LIN {X 0,Y 424.552,Z 355.445,A -85,B 0,C 180,E1 -10322.013,E2 -10322.013} C_VEL
LIN {X 0,Y 427.893,Z 370.379,A -85,B 0,C 180,E1 -10322.491,E2 -10322.491} C_VEL
LIN {X 0,Y 426.261,Z 483.338,A -85,B 0,C 180,E1 -10324.453,E2 -10324.453} C_VEL
LIN {X 0,Y 425.683,Z 497.997,A -85,B 0,C 180,E1 -10324.903,E2 -10324.903} C_VEL
LIN {X 0,Y 424.866,Z 511.461,A -85,B 0,C 180,E1 -10325.503,E2 -10325.503} C_VEL
LIN {X 0,Y 424.074,Z 524.723,A -85,B 0,C 180,E1 -10326.304,E2 -10326.304} C_VEL
LIN {X 0,Y 423.002,Z 537.419,A -85,B 0,C 180,E1 -10327.276,E2 -10327.276} C_VEL
LIN {X 0,Y 421.99,Z 548.966,A -85,B 0,C 180,E1 -10328.378,E2 -10328.378} C_VEL
LIN {X 0,Y 420.973,Z 560.52,A -85,B 0,C 180,E1 -10329.732,E2 -10329.732} C_VEL
LIN {X 0,Y 419.941,Z 570.774,A -85,B 0,C 180,E1 -10331.206,E2 -10331.206} C_VEL
LIN {X 0,Y 419.14,Z 579.23,A -85,B 0,C 180,E1 -10332.682,E2 -10332.682} C_VEL
LIN {X 0,Y 418.394,Z 587.297,A -85,B 0,C 180,E1 -10334.409,E2 -10334.409} C_VEL
LIN {X 0,Y 418.003,Z 591.69,A -85,B 0,C 180,E1 -10335.539,E2 -10335.539} C_VEL
LIN {X 0,Y 417.168,Z 594.262,A -85,B 0,C 180,E1 -10336.26,E2 -10336.26} C_VEL
LIN {X 0,Y 414.047,Z 598.094,A -85,B 0,C 180,E1 -10337.445,E2 -10337.445} C_VEL
LIN {X 0,Y 411.436,Z 600.721,A -85,B 0,C 180,E1 -10338.424,E2 -10338.424} C_VEL
LIN {X 0,Y 410.257,Z 602.444,A -85,B 0,C 180,E1 -10339.2,E2 -10339.2} C_VEL
LIN {X 0,Y 410.128,Z 602.917,A -85,B 0,C 180,E1 -10339.467,E2 -10339.467} C_VEL
LIN {X 0,Y 409.996,Z 605.551,A -85,B 0,C 180,E1 -10341.125,E2 -10341.125} C_VEL
LIN {X 0,Y 409.948,Z 607.379,A -85,B 0,C 180,E1 -10343.108,E2 -10343.108} C_VEL
LIN {X 0,Y 409.945,Z 607.876,A -85,B 0,C 180,E1 -10345.083,E2 -10345.083} C_VEL
LIN {X 0,Y 409.955,Z 607.058,A -85,B 0,C 180,E1 -10347.052,E2 -10347.052} C_VEL
LIN {X 0,Y 410.017,Z 606.153,A -85,B 0,C 180,E1 -10348.035,E2 -10348.035} C_VEL
LIN {X 0,Y 409.997,Z 603.337,A -85,B 0,C 180,E1 -10350,E2 -10350} C_VEL
LIN {X 0,Y 410.238,Z 600.322,A -85,B 0,C 180,E1 -10351.472,E2 -10351.472} C_VEL
LIN {X 0,Y 410.609,Z 594.902,A -85,B 0,C 180,E1 -10353.434,E2 -10353.434} C_VEL
LIN {X 0,Y 411.027,Z 589.771,A -85,B 0,C 180,E1 -10354.904,E2 -10354.904} C_VEL
LIN {X 0,Y 411.731,Z 582.375,A -85,B 0,C 180,E1 -10356.616,E2 -10356.616} C_VEL
LIN {X 0,Y 412.149,Z 576.039,A -85,B 0,C 180,E1 -10357.841,E2 -10357.841} C_VEL
LIN {X 0,Y 412.694,Z 568.684,A -85,B 0,C 180,E1 -10359.063,E2 -10359.063} C_VEL
LIN {X 0,Y 413.77,Z 558.137,A -85,B 0,C 180,E1 -10360.521,E2 -10360.521} C_VEL
LIN {X 0,Y 414.662,Z 547.501,A -85,B 0,C 180,E1 -10361.735,E2 -10361.735} C_VEL
LIN {X 0,Y 415.578,Z 535.885,A -85,B 0,C 180,E1 -10362.824,E2 -10362.824} C_VEL
LIN {X 0,Y 416.477,Z 523.1,A -85,B 0,C 180,E1 -10363.79,E2 -10363.79} C_VEL
LIN {X 0,Y 417.318,Z 509.784,A -85,B 0,C 180,E1 -10364.57,E2 -10364.57} C_VEL
LIN {X 0,Y 417.971,Z 495.947,A -85,B 0,C 180,E1 -10365.17,E2 -10365.17} C_VEL
LIN {X 0,Y 418.364,Z 482.792,A -85,B 0,C 180,E1 -10365.561,E2 -10365.561} C_VEL
LIN {X 0,Y 419.945,Z 370.675,A -85,B 0,C 180,E1 -10367.508,E2 -10367.508} C_VEL
LIN {X 0,Y 415.529,Z 350.853,A -85,B 0,C 180,E1 -10368.102,E2 -10368.102} C_VEL
LIN {X 0,Y 414.038,Z 346.546,A -85,B 0,C 180,E1 -10368.292,E2 -10368.292} C_VEL
LIN {X 0,Y 411.331,Z 333.524,A -85,B 0,C 180,E1 -10371.289,E2 -10371.289} C_VEL
LIN {X 0,Y 411.216,Z 332.89,A -85,B 0,C 180,E1 -10371.493,E2 -10371.493} C_VEL
LIN {X 0,Y 411.19,Z 332.895,A -85,B 0,C 180,E1 -10375.058,E2 -10375.058} C_VEL
LIN {X 0,Y 411.171,Z 332.896,A -85,B 0,C 180,E1 -10378.594,E2 -10378.594} C_VEL
LIN {X 0,Y 411.156,Z 332.893,A -85,B 0,C 180,E1 -10381.998,E2 -10381.998} C_VEL
LIN {X 0,Y 411.202,Z 332.89,A -85,B 0,C 180,E1 -10384.876,E2 -10384.876} C_VEL
LIN {X 0,Y 411.188,Z 332.889,A -85,B 0,C 180,E1 -10388.165,E2 -10388.165} C_VEL
LIN {X 0,Y 411.161,Z 332.889,A -85,B 0,C 180,E1 -10391.808,E2 -10391.808} C_VEL
LIN {X 0,Y 411.176,Z 332.887,A -85,B 0,C 180,E1 -10395.509,E2 -10395.509} C_VEL
LIN {X 0,Y 411.148,Z 332.894,A -85,B 0,C 180,E1 -10398.775,E2 -10398.775} C_VEL
LIN {X 0,Y 411.18,Z 332.889,A -85,B 0,C 180,E1 -10402.024,E2 -10402.024} C_VEL
LIN {X 0,Y 411.204,Z 332.887,A -85,B 0,C 180,E1 -10405.123,E2 -10405.123} C_VEL
LIN {X 0,Y 411.162,Z 332.886,A -85,B 0,C 180,E1 -10408.002,E2 -10408.002} C_VEL
LIN {X 0,Y 411.172,Z 332.887,A -85,B 0,C 180,E1 -10411.406,E2 -10411.406} C_VEL
LIN {X 0,Y 411.191,Z 332.889,A -85,B 0,C 180,E1 -10414.941,E2 -10414.941} C_VEL
LIN {X 0,Y 411.205,Z 332.883,A -85,B 0,C 180,E1 -10417.913,E2 -10417.913} C_VEL
LIN {X 0,Y 411.216,Z 332.876,A -85,B 0,C 180,E1 -10421.051,E2 -10421.051} C_VEL
LIN {X 0,Y 411.213,Z 332.889,A -85,B 0,C 180,E1 -10424.13,E2 -10424.13} C_VEL
LIN {X 0,Y 411.307,Z 332.864,A -85,B 0,C 180,E1 -10427.165,E2 -10427.165} C_VEL
LIN {X 0,Y 411.293,Z 332.86,A -85,B 0,C 180,E1 -10430.161,E2 -10430.161} C_VEL
LIN {X 0,Y 411.395,Z 332.861,A -85,B 0,C 180,E1 -10433.132,E2 -10433.132} C_VEL
LIN {X 0,Y 411.299,Z 332.872,A -85,B 0,C 180,E1 -10435.099,E2 -10435.099} C_VEL
LIN {X 0,Y 411.512,Z 332.851,A -85,B 0,C 180,E1 -10438.042,E2 -10438.042} C_VEL
LIN {X 0,Y 411.44,Z 332.851,A -85,B 0,C 180,E1 -10440.978,E2 -10440.978} C_VEL
LIN {X 0,Y 411.434,Z 332.857,A -85,B 0,C 180,E1 -10442.937,E2 -10442.937} C_VEL
LIN {X 0,Y 411.436,Z 332.857,A -85,B 0,C 180,E1 -10445.882,E2 -10445.882} C_VEL
LIN {X 0,Y 411.321,Z 332.87,A -85,B 0,C 180,E1 -10448.846,E2 -10448.846} C_VEL
LIN {X 0,Y 411.286,Z 332.879,A -85,B 0,C 180,E1 -10451.832,E2 -10451.832} C_VEL
LIN {X 0,Y 411.262,Z 332.876,A -85,B 0,C 180,E1 -10454.852,E2 -10454.852} C_VEL
LIN {X 0,Y 411.253,Z 332.882,A -85,B 0,C 180,E1 -10457.915,E2 -10457.915} C_VEL
LIN {X 0,Y 411.199,Z 332.886,A -85,B 0,C 180,E1 -10461.034,E2 -10461.034} C_VEL
LIN {X 0,Y 411.22,Z 332.886,A -85,B 0,C 180,E1 -10464.216,E2 -10464.216} C_VEL
LIN {X 0,Y 411.243,Z 332.885,A -85,B 0,C 180,E1 -10467.479,E2 -10467.479} C_VEL
LIN {X 0,Y 411.191,Z 332.889,A -85,B 0,C 180,E1 -10470.847,E2 -10470.847} C_VEL
LIN {X 0,Y 411.208,Z 332.888,A -85,B 0,C 180,E1 -10474.333,E2 -10474.333} C_VEL
LIN {X 0,Y 411.202,Z 332.889,A -85,B 0,C 180,E1 -10477.973,E2 -10477.973} C_VEL
LIN {X 0,Y 411.185,Z 332.89,A -85,B 0,C 180,E1 -10480.504,E2 -10480.504} C_VEL
LIN {X 0,Y 411.175,Z 332.894,A -85,B 0,C 180,E1 -10483.133,E2 -10483.133} C_VEL
LIN {X 0,Y 411.169,Z 332.894,A -85,B 0,C 180,E1 -10485.881,E2 -10485.881} C_VEL
LIN {X 0,Y 411.164,Z 332.892,A -85,B 0,C 180,E1 -10488.771,E2 -10488.771} C_VEL
LIN {X 0,Y 411.2,Z 332.893,A -85,B 0,C 180,E1 -10492.027,E2 -10492.027} C_VEL
LIN {X 0,Y 411.207,Z 332.893,A -85,B 0,C 180,E1 -10495.666,E2 -10495.666} C_VEL
LIN {X 0,Y 411.192,Z 332.892,A -85,B 0,C 180,E1 -10499.152,E2 -10499.152} C_VEL
LIN {X 0,Y 411.25,Z 333.05,A -85,B 0,C 180,E1 -10500.009,E2 -10500.009} C_VEL
LIN {X 0,Y 414.199,Z 346.153,A -85,B 0,C 180,E1 -10502.734,E2 -10502.734} C_VEL
LIN {X 0,Y 415.494,Z 353.398,A -85,B 0,C 180,E1 -10504.179,E2 -10504.179} C_VEL
LIN {X 0,Y 414.54,Z 367.529,A -85,B 0,C 180,E1 -10506.768,E2 -10506.768} C_VEL
LIN {X 0,Y 419.74,Z 398.333,A -85,B 0,C 180,E1 -10507.617,E2 -10507.617} C_VEL
LIN {X 0,Y 418.158,Z 504.873,A -85,B 0,C 180,E1 -10509.461,E2 -10509.461} C_VEL
LIN {X 0,Y 417.629,Z 519.149,A -85,B 0,C 180,E1 -10509.883,E2 -10509.883} C_VEL
LIN {X 0,Y 416.866,Z 532.72,A -85,B 0,C 180,E1 -10510.475,E2 -10510.475} C_VEL
LIN {X 0,Y 415.995,Z 546.287,A -85,B 0,C 180,E1 -10511.277,E2 -10511.277} C_VEL
LIN {X 0,Y 415.02,Z 559.153,A -85,B 0,C 180,E1 -10512.253,E2 -10512.253} C_VEL
LIN {X 0,Y 413.988,Z 570.843,A -85,B 0,C 180,E1 -10513.353,E2 -10513.353} C_VEL
LIN {X 0,Y 412.966,Z 582.538,A -85,B 0,C 180,E1 -10514.705,E2 -10514.705} C_VEL
LIN {X 0,Y 412.077,Z 592.992,A -85,B 0,C 180,E1 -10516.186,E2 -10516.186} C_VEL
LIN {X 0,Y 411.388,Z 601.614,A -85,B 0,C 180,E1 -10517.67,E2 -10517.67} C_VEL
LIN {X 0,Y 410.758,Z 609.847,A -85,B 0,C 180,E1 -10519.401,E2 -10519.401} C_VEL
LIN {X 0,Y 410.344,Z 616.475,A -85,B 0,C 180,E1 -10521.133,E2 -10521.133} C_VEL
LIN {X 0,Y 410.158,Z 622.354,A -85,B 0,C 180,E1 -10523.111,E2 -10523.111} C_VEL
LIN {X 0,Y 409.988,Z 626.639,A -85,B 0,C 180,E1 -10525.083,E2 -10525.083} C_VEL
LIN {X 0,Y 409.923,Z 629.47,A -85,B 0,C 180,E1 -10527.052,E2 -10527.052} C_VEL
LIN {X 0,Y 409.933,Z 630.928,A -85,B 0,C 180,E1 -10529.018,E2 -10529.018} C_VEL
LIN {X 0,Y 409.933,Z 631.045,A -85,B 0,C 180,E1 -10530.982,E2 -10530.982} C_VEL
LIN {X 0,Y 409.92,Z 629.831,A -85,B 0,C 180,E1 -10532.948,E2 -10532.948} C_VEL
LIN {X 0,Y 409.988,Z 627.259,A -85,B 0,C 180,E1 -10534.917,E2 -10534.917} C_VEL
LIN {X 0,Y 410.156,Z 623.241,A -85,B 0,C 180,E1 -10536.889,E2 -10536.889} C_VEL
LIN {X 0,Y 410.4,Z 617.672,A -85,B 0,C 180,E1 -10538.866,E2 -10538.866} C_VEL
LIN {X 0,Y 410.797,Z 611.402,A -85,B 0,C 180,E1 -10540.598,E2 -10540.598} C_VEL
LIN {X 0,Y 411.586,Z 603.609,A -85,B 0,C 180,E1 -10542.324,E2 -10542.324} C_VEL
LIN {X 0,Y 412.228,Z 595.485,A -85,B 0,C 180,E1 -10543.809,E2 -10543.809} C_VEL
LIN {X 0,Y 413.194,Z 585.715,A -85,B 0,C 180,E1 -10545.286,E2 -10545.286} C_VEL
LIN {X 0,Y 414.288,Z 574.884,A -85,B 0,C 180,E1 -10546.635,E2 -10546.635} C_VEL
LIN {X 0,Y 415.564,Z 562.897,A -85,B 0,C 180,E1 -10547.85,E2 -10547.85} C_VEL
LIN {X 0,Y 416.547,Z 551.215,A -85,B 0,C 180,E1 -10548.816,E2 -10548.816} C_VEL
LIN {X 0,Y 417.55,Z 538.211,A -85,B 0,C 180,E1 -10549.672,E2 -10549.672} C_VEL
LIN {X 0,Y 418.434,Z 524.264,A -85,B 0,C 180,E1 -10550.365,E2 -10550.365} C_VEL
LIN {X 0,Y 419.169,Z 510.595,A -85,B 0,C 180,E1 -10550.84,E2 -10550.84} C_VEL
LIN {X 0,Y 419.577,Z 495.358,A -85,B 0,C 180,E1 -10551.173,E2 -10551.173} C_VEL
LIN {X 0,Y 421.022,Z 397.613,A -85,B 0,C 180,E1 -10552.873,E2 -10552.873} C_VEL
LIN {X 0,Y 417.283,Z 377.293,A -85,B 0,C 180,E1 -10553.484,E2 -10553.484} C_VEL
LIN {X 0,Y 415.256,Z 367.358,A -85,B 0,C 180,E1 -10553.827,E2 -10553.827} C_VEL
LIN {X 0,Y 416.244,Z 355.506,A -85,B 0,C 180,E1 -10556.04,E2 -10556.04} C_VEL
LIN {X 0,Y 414.321,Z 345.621,A -85,B 0,C 180,E1 -10558.108,E2 -10558.108} C_VEL
LIN {X 0,Y 411.205,Z 332.882,A -85,B 0,C 180,E1 -10560.955,E2 -10560.955} C_VEL
LIN {X 0,Y 411.207,Z 332.89,A -85,B 0,C 180,E1 -10564.334,E2 -10564.334} C_VEL
LIN {X 0,Y 411.195,Z 332.887,A -85,B 0,C 180,E1 -10567.974,E2 -10567.974} C_VEL
LIN {X 0,Y 411.165,Z 332.891,A -85,B 0,C 180,E1 -10571.229,E2 -10571.229} C_VEL
LIN {X 0,Y 411.177,Z 332.895,A -85,B 0,C 180,E1 -10574.491,E2 -10574.491} C_VEL
LIN {X 0,Y 411.179,Z 332.89,A -85,B 0,C 180,E1 -10578.195,E2 -10578.195} C_VEL
LIN {X 0,Y 411.224,Z 332.883,A -85,B 0,C 180,E1 -10580.777,E2 -10580.777} C_VEL
LIN {X 0,Y 411.199,Z 332.89,A -85,B 0,C 180,E1 -10584.472,E2 -10584.472} C_VEL
LIN {X 0,Y 411.209,Z 332.885,A -85,B 0,C 180,E1 -10586.874,E2 -10586.874} C_VEL
LIN {X 0,Y 411.215,Z 332.887,A -85,B 0,C 180,E1 -10590.65,E2 -10590.65} C_VEL
LIN {X 0,Y 411.198,Z 332.885,A -85,B 0,C 180,E1 -10593.617,E2 -10593.617} C_VEL
LIN {X 0,Y 411.199,Z 332.884,A -85,B 0,C 180,E1 -10596.852,E2 -10596.852} C_VEL
LIN {X 0,Y 411.218,Z 332.889,A -85,B 0,C 180,E1 -10600.051,E2 -10600.051} C_VEL
LIN {X 0,Y 411.266,Z 332.875,A -85,B 0,C 180,E1 -10603.132,E2 -10603.132} C_VEL
LIN {X 0,Y 411.309,Z 332.866,A -85,B 0,C 180,E1 -10606.896,E2 -10606.896} C_VEL
LIN {X 0,Y 411.294,Z 332.876,A -85,B 0,C 180,E1 -10610.162,E2 -10610.162} C_VEL
LIN {X 0,Y 411.396,Z 332.86,A -85,B 0,C 180,E1 -10613.132,E2 -10613.132} C_VEL
LIN {X 0,Y 411.298,Z 332.874,A -85,B 0,C 180,E1 -10615.099,E2 -10615.099} C_VEL
LIN {X 0,Y 411.506,Z 332.85,A -85,B 0,C 180,E1 -10618.043,E2 -10618.043} C_VEL
LIN {X 0,Y 411.381,Z 332.86,A -85,B 0,C 180,E1 -10620.979,E2 -10620.979} C_VEL
LIN {X 0,Y 411.45,Z 332.852,A -85,B 0,C 180,E1 -10622.938,E2 -10622.938} C_VEL
LIN {X 0,Y 411.394,Z 332.854,A -85,B 0,C 180,E1 -10626.478,E2 -10626.478} C_VEL
LIN {X 0,Y 411.321,Z 332.871,A -85,B 0,C 180,E1 -10628.846,E2 -10628.846} C_VEL
LIN {X 0,Y 411.287,Z 332.873,A -85,B 0,C 180,E1 -10631.833,E2 -10631.833} C_VEL
LIN {X 0,Y 411.234,Z 332.882,A -85,B 0,C 180,E1 -10634.854,E2 -10634.854} C_VEL
LIN {X 0,Y 411.198,Z 332.891,A -85,B 0,C 180,E1 -10637.918,E2 -10637.918} C_VEL
LIN {X 0,Y 411.19,Z 332.883,A -85,B 0,C 180,E1 -10641.035,E2 -10641.035} C_VEL
LIN {X 0,Y 411.194,Z 332.884,A -85,B 0,C 180,E1 -10644.218,E2 -10644.218} C_VEL
LIN {X 0,Y 411.148,Z 332.896,A -85,B 0,C 180,E1 -10647.486,E2 -10647.486} C_VEL
LIN {X 0,Y 411.195,Z 332.87,A -85,B 0,C 180,E1 -10649.714,E2 -10649.714} C_VEL
LIN {X 0,Y 411.207,Z 332.887,A -85,B 0,C 180,E1 -10653.156,E2 -10653.156} C_VEL
LIN {X 0,Y 411.191,Z 332.873,A -85,B 0,C 180,E1 -10656.552,E2 -10656.552} C_VEL
LIN {X 0,Y 411.166,Z 332.892,A -85,B 0,C 180,E1 -10659.719,E2 -10659.719} C_VEL
LIN {X 0,Y 411.164,Z 332.894,A -85,B 0,C 180,E1 -10663.135,E2 -10663.135} C_VEL
LIN {X 0,Y 411.166,Z 332.887,A -85,B 0,C 180,E1 -10665.882,E2 -10665.882} C_VEL
LIN {X 0,Y 411.159,Z 332.892,A -85,B 0,C 180,E1 -10669.493,E2 -10669.493} C_VEL
LIN {X 0,Y 411.18,Z 332.894,A -85,B 0,C 180,E1 -10672.024,E2 -10672.024} C_VEL
LIN {X 0,Y 411.203,Z 332.891,A -85,B 0,C 180,E1 -10675.124,E2 -10675.124} C_VEL
LIN {X 0,Y 411.194,Z 332.982,A -85,B 0,C 180,E1 -10677.824,E2 -10677.824} C_VEL
LIN {X 0,Y 413.974,Z 345.407,A -85,B 0,C 180,E1 -10680.845,E2 -10680.845} C_VEL
LIN {X 0,Y 414.26,Z 346.859,A -85,B 0,C 180,E1 -10681.187,E2 -10681.187} C_VEL
LIN {X 0,Y 418.374,Z 357.743,A -85,B 0,C 180,E1 -10681.662,E2 -10681.662} C_VEL
LIN {X 0,Y 421.433,Z 371.468,A -85,B 0,C 180,E1 -10682.111,E2 -10682.111} C_VEL
LIN {X 0,Y 419.706,Z 483.714,A -85,B 0,C 180,E1 -10684.091,E2 -10684.091} C_VEL
LIN {X 0,Y 419.168,Z 497.624,A -85,B 0,C 180,E1 -10684.522,E2 -10684.522} C_VEL
LIN {X 0,Y 418.25,Z 511.823,A -85,B 0,C 180,E1 -10685.16,E2 -10685.16} C_VEL
LIN {X 0,Y 417.46,Z 524.434,A -85,B 0,C 180,E1 -10685.93,E2 -10685.93} C_VEL
LIN {X 0,Y 416.379,Z 536.951,A -85,B 0,C 180,E1 -10686.894,E2 -10686.894} C_VEL
LIN {X 0,Y 415.297,Z 548.614,A -85,B 0,C 180,E1 -10688.011,E2 -10688.011} C_VEL
LIN {X 0,Y 414.22,Z 560.262,A -85,B 0,C 180,E1 -10689.386,E2 -10689.386} C_VEL
LIN {X 0,Y 413.113,Z 570.622,A -85,B 0,C 180,E1 -10690.884,E2 -10690.884} C_VEL
LIN {X 0,Y 412.263,Z 579.001,A -85,B 0,C 180,E1 -10692.357,E2 -10692.357} C_VEL
LIN {X 0,Y 411.454,Z 587.259,A -85,B 0,C 180,E1 -10694.139,E2 -10694.139} C_VEL
LIN {X 0,Y 410.91,Z 592.955,A -85,B 0,C 180,E1 -10695.641,E2 -10695.641} C_VEL
LIN {X 0,Y 410.441,Z 598.367,A -85,B 0,C 180,E1 -10697.428,E2 -10697.428} C_VEL
LIN {X 0,Y 410.128,Z 602.917,A -85,B 0,C 180,E1 -10699.467,E2 -10699.467} C_VEL
LIN {X 0,Y 409.345,Z 604.353,A -85,B 0,C 180,E1 -10700.263,E2 -10700.263} C_VEL
LIN {X 0,Y 406.37,Z 606.202,A -85,B 0,C 180,E1 -10701.567,E2 -10701.567} C_VEL
LIN {X 0,Y 403.952,Z 607.261,A -85,B 0,C 180,E1 -10702.629,E2 -10702.629} C_VEL
LIN {X 0,Y 402.973,Z 607.773,A -85,B 0,C 180,E1 -10703.456,E2 -10703.456} C_VEL
LIN {X 0,Y 402.923,Z 607.901,A -85,B 0,C 180,E1 -10703.736,E2 -10703.736} C_VEL
LIN {X 0,Y 402.861,Z 608.087,A -85,B 0,C 180,E1 -10704.996,E2 -10704.996} C_VEL
LIN {X 0,Y 402.852,Z 607.307,A -85,B 0,C 180,E1 -10707,E2 -10707} C_VEL
LIN {X 0,Y 402.927,Z 606.42,A -85,B 0,C 180,E1 -10708.001,E2 -10708.001} C_VEL
LIN {X 0,Y 402.918,Z 603.642,A -85,B 0,C 180,E1 -10710,E2 -10710} C_VEL
LIN {X 0,Y 403.158,Z 600.662,A -85,B 0,C 180,E1 -10711.498,E2 -10711.498} C_VEL
LIN {X 0,Y 403.535,Z 595.292,A -85,B 0,C 180,E1 -10713.495,E2 -10713.495} C_VEL
LIN {X 0,Y 403.991,Z 590.187,A -85,B 0,C 180,E1 -10714.99,E2 -10714.99} C_VEL
LIN {X 0,Y 404.722,Z 582.857,A -85,B 0,C 180,E1 -10716.731,E2 -10716.731} C_VEL
LIN {X 0,Y 405.321,Z 575.069,A -85,B 0,C 180,E1 -10718.251,E2 -10718.251} C_VEL
LIN {X 0,Y 405.72,Z 569.26,A -85,B 0,C 180,E1 -10719.22,E2 -10719.22} C_VEL
LIN {X 0,Y 406.829,Z 558.787,A -85,B 0,C 180,E1 -10720.702,E2 -10720.702} C_VEL
LIN {X 0,Y 407.83,Z 547.083,A -85,B 0,C 180,E1 -10722.061,E2 -10722.061} C_VEL
LIN {X 0,Y 408.808,Z 535.33,A -85,B 0,C 180,E1 -10723.167,E2 -10723.167} C_VEL
LIN {X 0,Y 409.78,Z 522.357,A -85,B 0,C 180,E1 -10724.146,E2 -10724.146} C_VEL
LIN {X 0,Y 410.674,Z 508.677,A -85,B 0,C 180,E1 -10724.938,E2 -10724.938} C_VEL
LIN {X 0,Y 411.293,Z 495.102,A -85,B 0,C 180,E1 -10725.517,E2 -10725.517} C_VEL
LIN {X 0,Y 411.669,Z 481.3,A -85,B 0,C 180,E1 -10725.915,E2 -10725.915} C_VEL
LIN {X 0,Y 413.28,Z 371.634,A -85,B 0,C 180,E1 -10727.845,E2 -10727.845} C_VEL
LIN {X 0,Y 409.258,Z 353.309,A -85,B 0,C 180,E1 -10728.403,E2 -10728.403} C_VEL
LIN {X 0,Y 406.919,Z 346.861,A -85,B 0,C 180,E1 -10728.665,E2 -10728.665} C_VEL
LIN {X 0,Y 404.149,Z 333.77,A -85,B 0,C 180,E1 -10731.754,E2 -10731.754} C_VEL
LIN {X 0,Y 404.155,Z 333.77,A -85,B 0,C 180,E1 -10735.277,E2 -10735.277} C_VEL
LIN {X 0,Y 404.15,Z 333.767,A -85,B 0,C 180,E1 -10739.138,E2 -10739.138} C_VEL
LIN {X 0,Y 404.138,Z 333.77,A -85,B 0,C 180,E1 -10742.622,E2 -10742.622} C_VEL
LIN {X 0,Y 404.145,Z 333.768,A -85,B 0,C 180,E1 -10745.182,E2 -10745.182} C_VEL
LIN {X 0,Y 404.13,Z 333.77,A -85,B 0,C 180,E1 -10748.76,E2 -10748.76} C_VEL
LIN {X 0,Y 404.107,Z 333.768,A -85,B 0,C 180,E1 -10751.596,E2 -10751.596} C_VEL
LIN {X 0,Y 404.145,Z 333.768,A -85,B 0,C 180,E1 -10754.521,E2 -10754.521} C_VEL
LIN {X 0,Y 404.122,Z 333.768,A -85,B 0,C 180,E1 -10757.293,E2 -10757.293} C_VEL
LIN {X 0,Y 404.136,Z 333.766,A -85,B 0,C 180,E1 -10759.951,E2 -10759.951} C_VEL
LIN {X 0,Y 404.133,Z 333.765,A -85,B 0,C 180,E1 -10763.126,E2 -10763.126} C_VEL
LIN {X 0,Y 404.14,Z 333.769,A -85,B 0,C 180,E1 -10766.187,E2 -10766.187} C_VEL
LIN {X 0,Y 404.142,Z 333.766,A -85,B 0,C 180,E1 -10769.714,E2 -10769.714} C_VEL
LIN {X 0,Y 404.105,Z 333.766,A -85,B 0,C 180,E1 -10773.116,E2 -10773.116} C_VEL
LIN {X 0,Y 404.152,Z 333.766,A -85,B 0,C 180,E1 -10776.424,E2 -10776.424} C_VEL
LIN {X 0,Y 404.159,Z 333.746,A -85,B 0,C 180,E1 -10779.888,E2 -10779.888} C_VEL
LIN {X 0,Y 404.176,Z 333.761,A -85,B 0,C 180,E1 -10783.013,E2 -10783.013} C_VEL
LIN {X 0,Y 404.287,Z 333.739,A -85,B 0,C 180,E1 -10786.939,E2 -10786.939} C_VEL
LIN {X 0,Y 404.259,Z 333.733,A -85,B 0,C 180,E1 -10789.988,E2 -10789.988} C_VEL
LIN {X 0,Y 404.345,Z 333.74,A -85,B 0,C 180,E1 -10793.011,E2 -10793.011} C_VEL
LIN {X 0,Y 404.27,Z 333.748,A -85,B 0,C 180,E1 -10795.013,E2 -10795.013} C_VEL
LIN {X 0,Y 404.481,Z 333.727,A -85,B 0,C 180,E1 -10798.008,E2 -10798.008} C_VEL
LIN {X 0,Y 404.405,Z 333.727,A -85,B 0,C 180,E1 -10800.995,E2 -10800.995} C_VEL
LIN {X 0,Y 404.394,Z 333.734,A -85,B 0,C 180,E1 -10802.988,E2 -10802.988} C_VEL
LIN {X 0,Y 404.384,Z 333.736,A -85,B 0,C 180,E1 -10805.985,E2 -10805.985} C_VEL
LIN {X 0,Y 404.268,Z 333.748,A -85,B 0,C 180,E1 -10809.001,E2 -10809.001} C_VEL
LIN {X 0,Y 404.259,Z 333.756,A -85,B 0,C 180,E1 -10812.041,E2 -10812.041} C_VEL
LIN {X 0,Y 404.209,Z 333.755,A -85,B 0,C 180,E1 -10815.118,E2 -10815.118} C_VEL
LIN {X 0,Y 404.211,Z 333.757,A -85,B 0,C 180,E1 -10818.238,E2 -10818.238} C_VEL
LIN {X 0,Y 404.142,Z 333.768,A -85,B 0,C 180,E1 -10821.419,E2 -10821.419} C_VEL
LIN {X 0,Y 404.169,Z 333.762,A -85,B 0,C 180,E1 -10824.666,E2 -10824.666} C_VEL
LIN {X 0,Y 404.188,Z 333.763,A -85,B 0,C 180,E1 -10828,E2 -10828} C_VEL
LIN {X 0,Y 404.141,Z 333.773,A -85,B 0,C 180,E1 -10831.558,E2 -10831.558} C_VEL
LIN {X 0,Y 404.187,Z 333.763,A -85,B 0,C 180,E1 -10835.016,E2 -10835.016} C_VEL
LIN {X 0,Y 404.161,Z 333.763,A -85,B 0,C 180,E1 -10838.756,E2 -10838.756} C_VEL
LIN {X 0,Y 404.125,Z 333.775,A -85,B 0,C 180,E1 -10841.6,E2 -10841.6} C_VEL
LIN {X 0,Y 404.146,Z 333.766,A -85,B 0,C 180,E1 -10844.522,E2 -10844.522} C_VEL
LIN {X 0,Y 404.137,Z 333.771,A -85,B 0,C 180,E1 -10847.295,E2 -10847.295} C_VEL
LIN {X 0,Y 404.17,Z 333.767,A -85,B 0,C 180,E1 -10849.955,E2 -10849.955} C_VEL
LIN {X 0,Y 404.141,Z 333.773,A -85,B 0,C 180,E1 -10853.124,E2 -10853.124} C_VEL
LIN {X 0,Y 404.146,Z 333.771,A -85,B 0,C 180,E1 -10856.188,E2 -10856.188} C_VEL
LIN {X 0,Y 404.186,Z 333.908,A -85,B 0,C 180,E1 -10859.682,E2 -10859.682} C_VEL
LIN {X 0,Y 407.188,Z 347.194,A -85,B 0,C 180,E1 -10862.503,E2 -10862.503} C_VEL
LIN {X 0,Y 408.587,Z 354.535,A -85,B 0,C 180,E1 -10864.002,E2 -10864.002} C_VEL
LIN {X 0,Y 407.712,Z 367.579,A -85,B 0,C 180,E1 -10866.415,E2 -10866.415} C_VEL
LIN {X 0,Y 413.05,Z 398.587,A -85,B 0,C 180,E1 -10867.275,E2 -10867.275} C_VEL
LIN {X 0,Y 411.45,Z 504.747,A -85,B 0,C 180,E1 -10869.143,E2 -10869.143} C_VEL
LIN {X 0,Y 410.894,Z 518.989,A -85,B 0,C 180,E1 -10869.572,E2 -10869.572} C_VEL
LIN {X 0,Y 410.057,Z 533.328,A -85,B 0,C 180,E1 -10870.215,E2 -10870.215} C_VEL
LIN {X 0,Y 409.243,Z 545.669,A -85,B 0,C 180,E1 -10870.956,E2 -10870.956} C_VEL
LIN {X 0,Y 408.224,Z 558.615,A -85,B 0,C 180,E1 -10871.947,E2 -10871.947} C_VEL
LIN {X 0,Y 407.113,Z 570.363,A -85,B 0,C 180,E1 -10873.063,E2 -10873.063} C_VEL
LIN {X 0,Y 406.228,Z 580.139,A -85,B 0,C 180,E1 -10874.188,E2 -10874.188} C_VEL
LIN {X 0,Y 405.199,Z 590.958,A -85,B 0,C 180,E1 -10875.69,E2 -10875.69} C_VEL
LIN {X 0,Y 404.562,Z 599.894,A -85,B 0,C 180,E1 -10877.203,E2 -10877.203} C_VEL
LIN {X 0,Y 403.83,Z 608.442,A -85,B 0,C 180,E1 -10878.963,E2 -10878.963} C_VEL
LIN {X 0,Y 403.387,Z 614.41,A -85,B 0,C 180,E1 -10880.473,E2 -10880.473} C_VEL
LIN {X 0,Y 403.063,Z 620.778,A -85,B 0,C 180,E1 -10882.486,E2 -10882.486} C_VEL
LIN {X 0,Y 402.965,Z 624.423,A -85,B 0,C 180,E1 -10883.993,E2 -10883.993} C_VEL
LIN {X 0,Y 402.84,Z 627.987,A -85,B 0,C 180,E1 -10885.998,E2 -10885.998} C_VEL
LIN {X 0,Y 402.877,Z 630.146,A -85,B 0,C 180,E1 -10888.001,E2 -10888.001} C_VEL
LIN {X 0,Y 402.849,Z 630.948,A -85,B 0,C 180,E1 -10890,E2 -10890} C_VEL
LIN {X 0,Y 402.862,Z 630.417,A -85,B 0,C 180,E1 -10892,E2 -10892} C_VEL
LIN {X 0,Y 402.839,Z 628.549,A -85,B 0,C 180,E1 -10894.002,E2 -10894.002} C_VEL
LIN {X 0,Y 402.945,Z 625.293,A -85,B 0,C 180,E1 -10896.007,E2 -10896.007} C_VEL
LIN {X 0,Y 403.142,Z 620.535,A -85,B 0,C 180,E1 -10898.017,E2 -10898.017} C_VEL
LIN {X 0,Y 403.589,Z 614.159,A -85,B 0,C 180,E1 -10900.029,E2 -10900.029} C_VEL
LIN {X 0,Y 404.242,Z 607.077,A -85,B 0,C 180,E1 -10901.788,E2 -10901.788} C_VEL
LIN {X 0,Y 404.95,Z 598.889,A -85,B 0,C 180,E1 -10903.444,E2 -10903.444} C_VEL
LIN {X 0,Y 405.941,Z 589.19,A -85,B 0,C 180,E1 -10905.052,E2 -10905.052} C_VEL
LIN {X 0,Y 407.137,Z 578.131,A -85,B 0,C 180,E1 -10906.548,E2 -10906.548} C_VEL
LIN {X 0,Y 408.37,Z 566.866,A -85,B 0,C 180,E1 -10907.787,E2 -10907.787} C_VEL
LIN {X 0,Y 409.583,Z 554.431,A -85,B 0,C 180,E1 -10908.898,E2 -10908.898} C_VEL
LIN {X 0,Y 410.632,Z 541.22,A -85,B 0,C 180,E1 -10909.838,E2 -10909.838} C_VEL
LIN {X 0,Y 411.569,Z 528.039,A -85,B 0,C 180,E1 -10910.556,E2 -10910.556} C_VEL
LIN {X 0,Y 412.433,Z 514.251,A -85,B 0,C 180,E1 -10911.099,E2 -10911.099} C_VEL
LIN {X 0,Y 412.999,Z 500.1,A -85,B 0,C 180,E1 -10911.461,E2 -10911.461} C_VEL
LIN {X 0,Y 414.579,Z 398.68,A -85,B 0,C 180,E1 -10913.258,E2 -10913.258} C_VEL
LIN {X 0,Y 410.897,Z 378.756,A -85,B 0,C 180,E1 -10913.873,E2 -10913.873} C_VEL
LIN {X 0,Y 408.54,Z 367.175,A -85,B 0,C 180,E1 -10914.273,E2 -10914.273} C_VEL
LIN {X 0,Y 409.384,Z 356.883,A -85,B 0,C 180,E1 -10916.235,E2 -10916.235} C_VEL
LIN {X 0,Y 407.351,Z 346.92,A -85,B 0,C 180,E1 -10918.37,E2 -10918.37} C_VEL
LIN {X 0,Y 404.18,Z 333.963,A -85,B 0,C 180,E1 -10921.297,E2 -10921.297} C_VEL
LIN {X 0,Y 404.146,Z 333.766,A -85,B 0,C 180,E1 -10923.812,E2 -10923.812} C_VEL
LIN {X 0,Y 404.138,Z 333.772,A -85,B 0,C 180,E1 -10926.875,E2 -10926.875} C_VEL
LIN {X 0,Y 404.149,Z 333.767,A -85,B 0,C 180,E1 -10930.08,E2 -10930.08} C_VEL
LIN {X 0,Y 404.154,Z 333.763,A -85,B 0,C 180,E1 -10933.084,E2 -10933.084} C_VEL
LIN {X 0,Y 404.15,Z 333.764,A -85,B 0,C 180,E1 -10935.926,E2 -10935.926} C_VEL
LIN {X 0,Y 404.121,Z 333.77,A -85,B 0,C 180,E1 -10938.635,E2 -10938.635} C_VEL
LIN {X 0,Y 404.157,Z 333.762,A -85,B 0,C 180,E1 -10941.492,E2 -10941.492} C_VEL
LIN {X 0,Y 404.186,Z 333.761,A -85,B 0,C 180,E1 -10944.984,E2 -10944.984} C_VEL
LIN {X 0,Y 404.145,Z 333.769,A -85,B 0,C 180,E1 -10948.554,E2 -10948.554} C_VEL
LIN {X 0,Y 404.159,Z 333.764,A -85,B 0,C 180,E1 -10950.863,E2 -10950.863} C_VEL
LIN {X 0,Y 404.153,Z 333.764,A -85,B 0,C 180,E1 -10954.232,E2 -10954.232} C_VEL
LIN {X 0,Y 404.171,Z 333.76,A -85,B 0,C 180,E1 -10957.508,E2 -10957.508} C_VEL
LIN {X 0,Y 404.168,Z 333.762,A -85,B 0,C 180,E1 -10960.708,E2 -10960.708} C_VEL
LIN {X 0,Y 404.225,Z 333.757,A -85,B 0,C 180,E1 -10963.849,E2 -10963.849} C_VEL
LIN {X 0,Y 404.286,Z 333.74,A -85,B 0,C 180,E1 -10966.939,E2 -10966.939} C_VEL
LIN {X 0,Y 404.259,Z 333.754,A -85,B 0,C 180,E1 -10969.989,E2 -10969.989} C_VEL
LIN {X 0,Y 404.346,Z 333.738,A -85,B 0,C 180,E1 -10973.012,E2 -10973.012} C_VEL
LIN {X 0,Y 404.269,Z 333.749,A -85,B 0,C 180,E1 -10975.014,E2 -10975.014} C_VEL
LIN {X 0,Y 404.475,Z 333.725,A -85,B 0,C 180,E1 -10978.009,E2 -10978.009} C_VEL
LIN {X 0,Y 404.352,Z 333.736,A -85,B 0,C 180,E1 -10980.996,E2 -10980.996} C_VEL
LIN {X 0,Y 404.408,Z 333.729,A -85,B 0,C 180,E1 -10982.989,E2 -10982.989} C_VEL
LIN {X 0,Y 404.347,Z 333.732,A -85,B 0,C 180,E1 -10986.472,E2 -10986.472} C_VEL
LIN {X 0,Y 404.268,Z 333.75,A -85,B 0,C 180,E1 -10989.002,E2 -10989.002} C_VEL
LIN {X 0,Y 404.26,Z 333.749,A -85,B 0,C 180,E1 -10992.042,E2 -10992.042} C_VEL
LIN {X 0,Y 404.179,Z 333.762,A -85,B 0,C 180,E1 -10995.119,E2 -10995.119} C_VEL
LIN {X 0,Y 404.149,Z 333.766,A -85,B 0,C 180,E1 -10998.241,E2 -10998.241} C_VEL
LIN {X 0,Y 404.134,Z 333.764,A -85,B 0,C 180,E1 -11001.42,E2 -11001.42} C_VEL
LIN {X 0,Y 404.139,Z 333.762,A -85,B 0,C 180,E1 -11004.669,E2 -11004.669} C_VEL
LIN {X 0,Y 404.104,Z 333.767,A -85,B 0,C 180,E1 -11008.007,E2 -11008.007} C_VEL
LIN {X 0,Y 404.143,Z 333.745,A -85,B 0,C 180,E1 -11010.286,E2 -11010.286} C_VEL
LIN {X 0,Y 404.141,Z 333.768,A -85,B 0,C 180,E1 -11013.813,E2 -11013.813} C_VEL
LIN {X 0,Y 404.133,Z 333.752,A -85,B 0,C 180,E1 -11016.874,E2 -11016.874} C_VEL
LIN {X 0,Y 404.12,Z 333.767,A -85,B 0,C 180,E1 -11020.075,E2 -11020.075} C_VEL
LIN {X 0,Y 404.144,Z 333.768,A -85,B 0,C 180,E1 -11023.082,E2 -11023.082} C_VEL
LIN {X 0,Y 404.123,Z 333.764,A -85,B 0,C 180,E1 -11025.922,E2 -11025.922} C_VEL
LIN {X 0,Y 404.103,Z 333.774,A -85,B 0,C 180,E1 -11028.633,E2 -11028.633} C_VEL
LIN {X 0,Y 404.136,Z 333.772,A -85,B 0,C 180,E1 -11031.496,E2 -11031.496} C_VEL
LIN {X 0,Y 404.174,Z 333.767,A -85,B 0,C 180,E1 -11034.982,E2 -11034.982} C_VEL
LIN {X 0,Y 404.196,Z 333.932,A -85,B 0,C 180,E1 -11037.446,E2 -11037.446} C_VEL
LIN {X 0,Y 407.12,Z 347.112,A -85,B 0,C 180,E1 -11040.704,E2 -11040.704} C_VEL
LIN {X 0,Y 412.098,Z 359.682,A -85,B 0,C 180,E1 -11041.285,E2 -11041.285} C_VEL
LIN {X 0,Y 414.996,Z 372.537,A -85,B 0,C 180,E1 -11041.719,E2 -11041.719} C_VEL
LIN {X 0,Y 413.184,Z 482.848,A -85,B 0,C 180,E1 -11043.685,E2 -11043.685} C_VEL
LIN {X 0,Y 412.635,Z 497.184,A -85,B 0,C 180,E1 -11044.122,E2 -11044.122} C_VEL
LIN {X 0,Y 411.786,Z 510.984,A -85,B 0,C 180,E1 -11044.743,E2 -11044.743} C_VEL
LIN {X 0,Y 410.88,Z 524.141,A -85,B 0,C 180,E1 -11045.544,E2 -11045.544} C_VEL
LIN {X 0,Y 409.767,Z 536.492,A -85,B 0,C 180,E1 -11046.499,E2 -11046.499} C_VEL
LIN {X 0,Y 408.552,Z 548.266,A -85,B 0,C 180,E1 -11047.629,E2 -11047.629} C_VEL
LIN {X 0,Y 407.663,Z 558.04,A -85,B 0,C 180,E1 -11048.775,E2 -11048.775} C_VEL
LIN {X 0,Y 406.461,Z 568.824,A -85,B 0,C 180,E1 -11050.295,E2 -11050.295} C_VEL
LIN {X 0,Y 405.486,Z 577.693,A -85,B 0,C 180,E1 -11051.821,E2 -11051.821} C_VEL
LIN {X 0,Y 404.733,Z 585.045,A -85,B 0,C 180,E1 -11053.35,E2 -11053.35} C_VEL
LIN {X 0,Y 404.096,Z 591.141,A -85,B 0,C 180,E1 -11054.878,E2 -11054.878} C_VEL
LIN {X 0,Y 403.683,Z 596.171,A -85,B 0,C 180,E1 -11056.406,E2 -11056.406} C_VEL
LIN {X 0,Y 403.222,Z 601.331,A -85,B 0,C 180,E1 -11058.437,E2 -11058.437} C_VEL
LIN {X 0,Y 402.967,Z 604.222,A -85,B 0,C 180,E1 -11059.956,E2 -11059.956} C_VEL
LIN {X 0,Y 402.869,Z 606.788,A -85,B 0,C 180,E1 -11061.978,E2 -11061.978} C_VEL
LIN {X 0,Y 402.923,Z 607.901,A -85,B 0,C 180,E1 -11063.736,E2 -11063.736} C_VEL
LIN {X 0,Y 402.329,Z 608.177,A -85,B 0,C 180,E1 -11064.569,E2 -11064.569} C_VEL
LIN {X 0,Y 399.482,Z 608.114,A -85,B 0,C 180,E1 -11065.924,E2 -11065.924} C_VEL
LIN {X 0,Y 397.012,Z 607.55,A -85,B 0,C 180,E1 -11067.016,E2 -11067.016} C_VEL
LIN {X 0,Y 395.925,Z 606.804,A -85,B 0,C 180,E1 -11067.855,E2 -11067.855} C_VEL
LIN {X 0,Y 395.826,Z 606.482,A -85,B 0,C 180,E1 -11068.138,E2 -11068.138} C_VEL
LIN {X 0,Y 395.841,Z 603.946,A -85,B 0,C 180,E1 -11070,E2 -11070} C_VEL
LIN {X 0,Y 396.046,Z 599.789,A -85,B 0,C 180,E1 -11072.034,E2 -11072.034} C_VEL
LIN {X 0,Y 396.593,Z 594.081,A -85,B 0,C 180,E1 -11074.065,E2 -11074.065} C_VEL
LIN {X 0,Y 397.206,Z 587.655,A -85,B 0,C 180,E1 -11075.839,E2 -11075.839} C_VEL
LIN {X 0,Y 397.803,Z 580.916,A -85,B 0,C 180,E1 -11077.359,E2 -11077.359} C_VEL
LIN {X 0,Y 398.423,Z 572.851,A -85,B 0,C 180,E1 -11078.879,E2 -11078.879} C_VEL
LIN {X 0,Y 399.502,Z 563.122,A -85,B 0,C 180,E1 -11080.388,E2 -11080.388} C_VEL
LIN {X 0,Y 400.565,Z 552.33,A -85,B 0,C 180,E1 -11081.769,E2 -11081.769} C_VEL
LIN {X 0,Y 401.537,Z 541.642,A -85,B 0,C 180,E1 -11082.895,E2 -11082.895} C_VEL
LIN {X 0,Y 402.467,Z 530.126,A -85,B 0,C 180,E1 -11083.893,E2 -11083.893} C_VEL
LIN {X 0,Y 403.415,Z 516.62,A -85,B 0,C 180,E1 -11084.825,E2 -11084.825} C_VEL
LIN {X 0,Y 404.179,Z 503.619,A -85,B 0,C 180,E1 -11085.506,E2 -11085.506} C_VEL
LIN {X 0,Y 404.74,Z 489.638,A -85,B 0,C 180,E1 -11086.034,E2 -11086.034} C_VEL
LIN {X 0,Y 405.099,Z 474.98,A -85,B 0,C 180,E1 -11086.375,E2 -11086.375} C_VEL
LIN {X 0,Y 406.679,Z 372.812,A -85,B 0,C 180,E1 -11088.185,E2 -11088.185} C_VEL
LIN {X 0,Y 402.827,Z 355.422,A -85,B 0,C 180,E1 -11088.73,E2 -11088.73} C_VEL
LIN {X 0,Y 399.723,Z 346.952,A -85,B 0,C 180,E1 -11089.104,E2 -11089.104} C_VEL
LIN {X 0,Y 397.123,Z 334.645,A -85,B 0,C 180,E1 -11092.056,E2 -11092.056} C_VEL
LIN {X 0,Y 397.097,Z 334.649,A -85,B 0,C 180,E1 -11095.494,E2 -11095.494} C_VEL
LIN {X 0,Y 397.063,Z 334.653,A -85,B 0,C 180,E1 -11098.548,E2 -11098.548} C_VEL
LIN {X 0,Y 397.077,Z 334.647,A -85,B 0,C 180,E1 -11101.834,E2 -11101.834} C_VEL
LIN {X 0,Y 397.118,Z 334.644,A -85,B 0,C 180,E1 -11104.494,E2 -11104.494} C_VEL
LIN {X 0,Y 397.088,Z 334.647,A -85,B 0,C 180,E1 -11108.277,E2 -11108.277} C_VEL
LIN {X 0,Y 397.048,Z 334.652,A -85,B 0,C 180,E1 -11110.914,E2 -11110.914} C_VEL
LIN {X 0,Y 397.089,Z 334.644,A -85,B 0,C 180,E1 -11113.65,E2 -11113.65} C_VEL
LIN {X 0,Y 397.093,Z 334.647,A -85,B 0,C 180,E1 -11116.523,E2 -11116.523} C_VEL
LIN {X 0,Y 397.087,Z 334.648,A -85,B 0,C 180,E1 -11120.419,E2 -11120.419} C_VEL
LIN {X 0,Y 397.095,Z 334.643,A -85,B 0,C 180,E1 -11123.004,E2 -11123.004} C_VEL
LIN {X 0,Y 397.101,Z 334.645,A -85,B 0,C 180,E1 -11126.287,E2 -11126.287} C_VEL
LIN {X 0,Y 397.075,Z 334.647,A -85,B 0,C 180,E1 -11129.117,E2 -11129.117} C_VEL
LIN {X 0,Y 397.063,Z 334.645,A -85,B 0,C 180,E1 -11132.252,E2 -11132.252} C_VEL
LIN {X 0,Y 397.106,Z 334.644,A -85,B 0,C 180,E1 -11134.865,E2 -11134.865} C_VEL
LIN {X 0,Y 397.097,Z 334.635,A -85,B 0,C 180,E1 -11138.181,E2 -11138.181} C_VEL
LIN {X 0,Y 397.116,Z 334.631,A -85,B 0,C 180,E1 -11141.424,E2 -11141.424} C_VEL
LIN {X 0,Y 397.127,Z 334.641,A -85,B 0,C 180,E1 -11144.606,E2 -11144.606} C_VEL
LIN {X 0,Y 397.222,Z 334.617,A -85,B 0,C 180,E1 -11147.742,E2 -11147.742} C_VEL
LIN {X 0,Y 397.239,Z 334.619,A -85,B 0,C 180,E1 -11150.838,E2 -11150.838} C_VEL
LIN {X 0,Y 397.333,Z 334.617,A -85,B 0,C 180,E1 -11153.908,E2 -11153.908} C_VEL
LIN {X 0,Y 397.45,Z 334.602,A -85,B 0,C 180,E1 -11157.973,E2 -11157.973} C_VEL
LIN {X 0,Y 397.37,Z 334.603,A -85,B 0,C 180,E1 -11161.013,E2 -11161.013} C_VEL
LIN {X 0,Y 397.328,Z 334.614,A -85,B 0,C 180,E1 -11163.042,E2 -11163.042} C_VEL
LIN {X 0,Y 397.335,Z 334.614,A -85,B 0,C 180,E1 -11166.092,E2 -11166.092} C_VEL
LIN {X 0,Y 397.238,Z 334.624,A -85,B 0,C 180,E1 -11169.162,E2 -11169.162} C_VEL
LIN {X 0,Y 397.222,Z 334.63,A -85,B 0,C 180,E1 -11172.258,E2 -11172.258} C_VEL
LIN {X 0,Y 397.182,Z 334.632,A -85,B 0,C 180,E1 -11175.392,E2 -11175.392} C_VEL
LIN {X 0,Y 397.163,Z 334.633,A -85,B 0,C 180,E1 -11178.573,E2 -11178.573} C_VEL
LIN {X 0,Y 397.1,Z 334.645,A -85,B 0,C 180,E1 -11181.818,E2 -11181.818} C_VEL
LIN {X 0,Y 397.126,Z 334.64,A -85,B 0,C 180,E1 -11185.133,E2 -11185.133} C_VEL
LIN {X 0,Y 397.152,Z 334.643,A -85,B 0,C 180,E1 -11187.773,E2 -11187.773} C_VEL
LIN {X 0,Y 397.08,Z 334.647,A -85,B 0,C 180,E1 -11190.882,E2 -11190.882} C_VEL
LIN {X 0,Y 397.127,Z 334.642,A -85,B 0,C 180,E1 -11194.493,E2 -11194.493} C_VEL
LIN {X 0,Y 397.108,Z 334.642,A -85,B 0,C 180,E1 -11198.274,E2 -11198.274} C_VEL
LIN {X 0,Y 397.091,Z 334.646,A -85,B 0,C 180,E1 -11200.908,E2 -11200.908} C_VEL
LIN {X 0,Y 397.102,Z 334.649,A -85,B 0,C 180,E1 -11203.648,E2 -11203.648} C_VEL
LIN {X 0,Y 397.103,Z 334.643,A -85,B 0,C 180,E1 -11206.521,E2 -11206.521} C_VEL
LIN {X 0,Y 397.115,Z 334.644,A -85,B 0,C 180,E1 -11210.423,E2 -11210.423} C_VEL
LIN {X 0,Y 397.11,Z 334.648,A -85,B 0,C 180,E1 -11214.265,E2 -11214.265} C_VEL
LIN {X 0,Y 397.116,Z 334.648,A -85,B 0,C 180,E1 -11216.727,E2 -11216.727} C_VEL
LIN {X 0,Y 397.127,Z 334.724,A -85,B 0,C 180,E1 -11219.335,E2 -11219.335} C_VEL
LIN {X 0,Y 400.175,Z 348.232,A -85,B 0,C 180,E1 -11222.264,E2 -11222.264} C_VEL
LIN {X 0,Y 401.575,Z 355.058,A -85,B 0,C 180,E1 -11223.693,E2 -11223.693} C_VEL
LIN {X 0,Y 401.463,Z 359.756,A -85,B 0,C 180,E1 -11224.602,E2 -11224.602} C_VEL
LIN {X 0,Y 400.843,Z 367.213,A -85,B 0,C 180,E1 -11226.012,E2 -11226.012} C_VEL
LIN {X 0,Y 406.366,Z 399.239,A -85,B 0,C 180,E1 -11226.929,E2 -11226.929} C_VEL
LIN {X 0,Y 404.896,Z 498.535,A -85,B 0,C 180,E1 -11228.689,E2 -11228.689} C_VEL
LIN {X 0,Y 404.406,Z 513.401,A -85,B 0,C 180,E1 -11229.063,E2 -11229.063} C_VEL
LIN {X 0,Y 403.633,Z 527.535,A -85,B 0,C 180,E1 -11229.62,E2 -11229.62} C_VEL
LIN {X 0,Y 402.823,Z 539.96,A -85,B 0,C 180,E1 -11230.295,E2 -11230.295} C_VEL
LIN {X 0,Y 401.822,Z 553.645,A -85,B 0,C 180,E1 -11231.264,E2 -11231.264} C_VEL
LIN {X 0,Y 400.613,Z 566.22,A -85,B 0,C 180,E1 -11232.385,E2 -11232.385} C_VEL
LIN {X 0,Y 399.53,Z 577.694,A -85,B 0,C 180,E1 -11233.653,E2 -11233.653} C_VEL
LIN {X 0,Y 398.616,Z 587.199,A -85,B 0,C 180,E1 -11234.926,E2 -11234.926} C_VEL
LIN {X 0,Y 397.801,Z 597.029,A -85,B 0,C 180,E1 -11236.509,E2 -11236.509} C_VEL
LIN {X 0,Y 397.022,Z 605.855,A -85,B 0,C 180,E1 -11238.254,E2 -11238.254} C_VEL
LIN {X 0,Y 396.437,Z 612.258,A -85,B 0,C 180,E1 -11239.789,E2 -11239.789} C_VEL
LIN {X 0,Y 396.129,Z 617.514,A -85,B 0,C 180,E1 -11241.326,E2 -11241.326} C_VEL
LIN {X 0,Y 395.986,Z 621.808,A -85,B 0,C 180,E1 -11242.863,E2 -11242.863} C_VEL
LIN {X 0,Y 395.822,Z 626.135,A -85,B 0,C 180,E1 -11244.907,E2 -11244.907} C_VEL
LIN {X 0,Y 395.725,Z 629.003,A -85,B 0,C 180,E1 -11246.946,E2 -11246.946} C_VEL
LIN {X 0,Y 395.789,Z 630.5,A -85,B 0,C 180,E1 -11248.983,E2 -11248.983} C_VEL
LIN {X 0,Y 395.789,Z 630.652,A -85,B 0,C 180,E1 -11251.017,E2 -11251.017} C_VEL
LIN {X 0,Y 395.721,Z 629.472,A -85,B 0,C 180,E1 -11253.054,E2 -11253.054} C_VEL
LIN {X 0,Y 395.802,Z 626.943,A -85,B 0,C 180,E1 -11255.094,E2 -11255.094} C_VEL
LIN {X 0,Y 395.989,Z 622.977,A -85,B 0,C 180,E1 -11257.137,E2 -11257.137} C_VEL
LIN {X 0,Y 396.294,Z 617.451,A -85,B 0,C 180,E1 -11259.184,E2 -11259.184} C_VEL
LIN {X 0,Y 396.784,Z 611.229,A -85,B 0,C 180,E1 -11260.977,E2 -11260.977} C_VEL
LIN {X 0,Y 397.606,Z 603.49,A -85,B 0,C 180,E1 -11262.765,E2 -11262.765} C_VEL
LIN {X 0,Y 398.382,Z 595.429,A -85,B 0,C 180,E1 -11264.299,E2 -11264.299} C_VEL
LIN {X 0,Y 399.461,Z 585.731,A -85,B 0,C 180,E1 -11265.825,E2 -11265.825} C_VEL
LIN {X 0,Y 400.689,Z 574.987,A -85,B 0,C 180,E1 -11267.217,E2 -11267.217} C_VEL
LIN {X 0,Y 402.023,Z 563.11,A -85,B 0,C 180,E1 -11268.473,E2 -11268.473} C_VEL
LIN {X 0,Y 403.183,Z 550.994,A -85,B 0,C 180,E1 -11269.513,E2 -11269.513} C_VEL
LIN {X 0,Y 404.313,Z 537.774,A -85,B 0,C 180,E1 -11270.41,E2 -11270.41} C_VEL
LIN {X 0,Y 405.276,Z 524.557,A -85,B 0,C 180,E1 -11271.09,E2 -11271.09} C_VEL
LIN {X 0,Y 406.069,Z 510.133,A -85,B 0,C 180,E1 -11271.612,E2 -11271.612} C_VEL
LIN {X 0,Y 406.532,Z 494.864,A -85,B 0,C 180,E1 -11271.953,E2 -11271.953} C_VEL
LIN {X 0,Y 408.161,Z 399.688,A -85,B 0,C 180,E1 -11273.656,E2 -11273.656} C_VEL
LIN {X 0,Y 404.066,Z 377.831,A -85,B 0,C 180,E1 -11274.353,E2 -11274.353} C_VEL
LIN {X 0,Y 401.805,Z 367.05,A -85,B 0,C 180,E1 -11274.727,E2 -11274.727} C_VEL
LIN {X 0,Y 402.511,Z 358.357,A -85,B 0,C 180,E1 -11276.418,E2 -11276.418} C_VEL
LIN {X 0,Y 400.424,Z 348.159,A -85,B 0,C 180,E1 -11278.65,E2 -11278.65} C_VEL
LIN {X 0,Y 397.425,Z 336.059,A -85,B 0,C 180,E1 -11281.445,E2 -11281.445} C_VEL
LIN {X 0,Y 397.083,Z 334.647,A -85,B 0,C 180,E1 -11281.837,E2 -11281.837} C_VEL
LIN {X 0,Y 397.127,Z 334.644,A -85,B 0,C 180,E1 -11284.493,E2 -11284.493} C_VEL
LIN {X 0,Y 397.103,Z 334.639,A -85,B 0,C 180,E1 -11288.275,E2 -11288.275} C_VEL
LIN {X 0,Y 397.09,Z 334.646,A -85,B 0,C 180,E1 -11290.909,E2 -11290.909} C_VEL
LIN {X 0,Y 397.102,Z 334.641,A -85,B 0,C 180,E1 -11293.649,E2 -11293.649} C_VEL
LIN {X 0,Y 397.104,Z 334.646,A -85,B 0,C 180,E1 -11296.521,E2 -11296.521} C_VEL
LIN {X 0,Y 397.116,Z 334.641,A -85,B 0,C 180,E1 -11300.423,E2 -11300.423} C_VEL
LIN {X 0,Y 397.11,Z 334.642,A -85,B 0,C 180,E1 -11304.266,E2 -11304.266} C_VEL
LIN {X 0,Y 397.117,Z 334.64,A -85,B 0,C 180,E1 -11306.727,E2 -11306.727} C_VEL
LIN {X 0,Y 397.121,Z 334.64,A -85,B 0,C 180,E1 -11310.296,E2 -11310.296} C_VEL
LIN {X 0,Y 397.098,Z 334.642,A -85,B 0,C 180,E1 -11313.739,E2 -11313.739} C_VEL
LIN {X 0,Y 397.107,Z 334.639,A -85,B 0,C 180,E1 -11317.086,E2 -11317.086} C_VEL
LIN {X 0,Y 397.151,Z 334.639,A -85,B 0,C 180,E1 -11320.353,E2 -11320.353} C_VEL
LIN {X 0,Y 397.17,Z 334.633,A -85,B 0,C 180,E1 -11323.554,E2 -11323.554} C_VEL
LIN {X 0,Y 397.232,Z 334.62,A -85,B 0,C 180,E1 -11326.703,E2 -11326.703} C_VEL
LIN {X 0,Y 397.219,Z 334.633,A -85,B 0,C 180,E1 -11329.809,E2 -11329.809} C_VEL
LIN {X 0,Y 397.298,Z 334.616,A -85,B 0,C 180,E1 -11332.887,E2 -11332.887} C_VEL
LIN {X 0,Y 397.24,Z 334.625,A -85,B 0,C 180,E1 -11334.925,E2 -11334.925} C_VEL
LIN {X 0,Y 397.444,Z 334.6,A -85,B 0,C 180,E1 -11337.974,E2 -11337.974} C_VEL
LIN {X 0,Y 397.322,Z 334.611,A -85,B 0,C 180,E1 -11341.014,E2 -11341.014} C_VEL
LIN {X 0,Y 397.342,Z 334.61,A -85,B 0,C 180,E1 -11343.042,E2 -11343.042} C_VEL
LIN {X 0,Y 397.304,Z 334.609,A -85,B 0,C 180,E1 -11346.465,E2 -11346.465} C_VEL
LIN {X 0,Y 397.238,Z 334.626,A -85,B 0,C 180,E1 -11349.163,E2 -11349.163} C_VEL
LIN {X 0,Y 397.223,Z 334.626,A -85,B 0,C 180,E1 -11352.258,E2 -11352.258} C_VEL
LIN {X 0,Y 397.127,Z 334.642,A -85,B 0,C 180,E1 -11355.394,E2 -11355.394} C_VEL
LIN {X 0,Y 397.097,Z 334.643,A -85,B 0,C 180,E1 -11358.577,E2 -11358.577} C_VEL
LIN {X 0,Y 397.094,Z 334.646,A -85,B 0,C 180,E1 -11361.819,E2 -11361.819} C_VEL
LIN {X 0,Y 397.106,Z 334.639,A -85,B 0,C 180,E1 -11365.135,E2 -11365.135} C_VEL
LIN {X 0,Y 397.064,Z 334.642,A -85,B 0,C 180,E1 -11368.549,E2 -11368.549} C_VEL
LIN {X 0,Y 397.08,Z 334.638,A -85,B 0,C 180,E1 -11371.835,E2 -11371.835} C_VEL
LIN {X 0,Y 397.12,Z 334.64,A -85,B 0,C 180,E1 -11374.494,E2 -11374.494} C_VEL
LIN {X 0,Y 397.089,Z 334.644,A -85,B 0,C 180,E1 -11378.277,E2 -11378.277} C_VEL
LIN {X 0,Y 397.053,Z 334.65,A -85,B 0,C 180,E1 -11381.976,E2 -11381.976} C_VEL
LIN {X 0,Y 397.087,Z 334.644,A -85,B 0,C 180,E1 -11385.069,E2 -11385.069} C_VEL
LIN {X 0,Y 397.053,Z 334.653,A -85,B 0,C 180,E1 -11388.024,E2 -11388.024} C_VEL
LIN {X 0,Y 397.09,Z 334.652,A -85,B 0,C 180,E1 -11391.147,E2 -11391.147} C_VEL
LIN {X 0,Y 397.1,Z 334.647,A -85,B 0,C 180,E1 -11394.502,E2 -11394.502} C_VEL
LIN {X 0,Y 397.153,Z 334.808,A -85,B 0,C 180,E1 -11397.033,E2 -11397.033} C_VEL
LIN {X 0,Y 399.958,Z 347.331,A -85,B 0,C 180,E1 -11400.199,E2 -11400.199} C_VEL
LIN {X 0,Y 405.974,Z 362.054,A -85,B 0,C 180,E1 -11400.913,E2 -11400.913} C_VEL
LIN {X 0,Y 408.578,Z 373.661,A -85,B 0,C 180,E1 -11401.314,E2 -11401.314} C_VEL
LIN {X 0,Y 406.661,Z 483.32,A -85,B 0,C 180,E1 -11403.299,E2 -11403.299} C_VEL
LIN {X 0,Y 406.088,Z 497.533,A -85,B 0,C 180,E1 -11403.743,E2 -11403.743} C_VEL
LIN {X 0,Y 405.276,Z 510.15,A -85,B 0,C 180,E1 -11404.308,E2 -11404.308} C_VEL
LIN {X 0,Y 404.419,Z 522.542,A -85,B 0,C 180,E1 -11405.051,E2 -11405.051} C_VEL
LIN {X 0,Y 403.329,Z 534.599,A -85,B 0,C 180,E1 -11405.964,E2 -11405.964} C_VEL
LIN {X 0,Y 402.056,Z 546.746,A -85,B 0,C 180,E1 -11407.112,E2 -11407.112} C_VEL
LIN {X 0,Y 400.945,Z 557.792,A -85,B 0,C 180,E1 -11408.401,E2 -11408.401} C_VEL
LIN {X 0,Y 399.862,Z 567.011,A -85,B 0,C 180,E1 -11409.688,E2 -11409.688} C_VEL
LIN {X 0,Y 398.785,Z 576.22,A -85,B 0,C 180,E1 -11411.238,E2 -11411.238} C_VEL
LIN {X 0,Y 397.812,Z 584.989,A -85,B 0,C 180,E1 -11413.052,E2 -11413.052} C_VEL
LIN {X 0,Y 397.124,Z 591.134,A -85,B 0,C 180,E1 -11414.606,E2 -11414.606} C_VEL
LIN {X 0,Y 396.53,Z 597.634,A -85,B 0,C 180,E1 -11416.679,E2 -11416.679} C_VEL
LIN {X 0,Y 396.109,Z 602.474,A -85,B 0,C 180,E1 -11418.745,E2 -11418.745} C_VEL
LIN {X 0,Y 395.828,Z 605.805,A -85,B 0,C 180,E1 -11420.805,E2 -11420.805} C_VEL
LIN {X 0,Y 395.777,Z 607.725,A -85,B 0,C 180,E1 -11422.859,E2 -11422.859} C_VEL
LIN {X 0,Y 395.78,Z 608.298,A -85,B 0,C 180,E1 -11424.906,E2 -11424.906} C_VEL
LIN {X 0,Y 395.751,Z 607.555,A -85,B 0,C 180,E1 -11426.946,E2 -11426.946} C_VEL
LIN {X 0,Y 395.826,Z 606.482,A -85,B 0,C 180,E1 -11428.138,E2 -11428.138} C_VEL
LIN {X 0,Y 395.12,Z 605.531,A -85,B 0,C 180,E1 -11428.975,E2 -11428.975} C_VEL
LIN {X 0,Y 392.258,Z 603.535,A -85,B 0,C 180,E1 -11430.328,E2 -11430.328} C_VEL
LIN {X 0,Y 389.555,Z 601.016,A -85,B 0,C 180,E1 -11431.681,E2 -11431.681} C_VEL
LIN {X 0,Y 389.113,Z 599.091,A -85,B 0,C 180,E1 -11432.506,E2 -11432.506} C_VEL
LIN {X 0,Y 389.549,Z 594.465,A -85,B 0,C 180,E1 -11434.138,E2 -11434.138} C_VEL
LIN {X 0,Y 390.097,Z 589.081,A -85,B 0,C 180,E1 -11435.687,E2 -11435.687} C_VEL
LIN {X 0,Y 390.74,Z 582.61,A -85,B 0,C 180,E1 -11437.233,E2 -11437.233} C_VEL
LIN {X 0,Y 391.413,Z 574.099,A -85,B 0,C 180,E1 -11438.913,E2 -11438.913} C_VEL
LIN {X 0,Y 392.363,Z 565.488,A -85,B 0,C 180,E1 -11440.319,E2 -11440.319} C_VEL
LIN {X 0,Y 393.456,Z 555.126,A -85,B 0,C 180,E1 -11441.723,E2 -11441.723} C_VEL
LIN {X 0,Y 394.545,Z 543.7,A -85,B 0,C 180,E1 -11442.996,E2 -11442.996} C_VEL
LIN {X 0,Y 395.633,Z 531.033,A -85,B 0,C 180,E1 -11444.138,E2 -11444.138} C_VEL
LIN {X 0,Y 396.544,Z 518.692,A -85,B 0,C 180,E1 -11445.023,E2 -11445.023} C_VEL
LIN {X 0,Y 397.425,Z 504.976,A -85,B 0,C 180,E1 -11445.777,E2 -11445.777} C_VEL
LIN {X 0,Y 398.048,Z 490.633,A -85,B 0,C 180,E1 -11446.344,E2 -11446.344} C_VEL
LIN {X 0,Y 398.446,Z 476.57,A -85,B 0,C 180,E1 -11446.689,E2 -11446.689} C_VEL
LIN {X 0,Y 400.057,Z 373.709,A -85,B 0,C 180,E1 -11448.544,E2 -11448.544} C_VEL
LIN {X 0,Y 396.523,Z 357.816,A -85,B 0,C 180,E1 -11449.054,E2 -11449.054} C_VEL
LIN {X 0,Y 392.561,Z 347.238,A -85,B 0,C 180,E1 -11449.514,E2 -11449.514} C_VEL
LIN {X 0,Y 390.084,Z 335.522,A -85,B 0,C 180,E1 -11452.406,E2 -11452.406} C_VEL
LIN {X 0,Y 390.053,Z 335.526,A -85,B 0,C 180,E1 -11455.722,E2 -11455.722} C_VEL
LIN {X 0,Y 390.024,Z 335.527,A -85,B 0,C 180,E1 -11459.113,E2 -11459.113} C_VEL
LIN {X 0,Y 390.041,Z 335.526,A -85,B 0,C 180,E1 -11462.722,E2 -11462.722} C_VEL
LIN {X 0,Y 390.043,Z 335.523,A -85,B 0,C 180,E1 -11465.822,E2 -11465.822} C_VEL
LIN {X 0,Y 390.036,Z 335.524,A -85,B 0,C 180,E1 -11469.211,E2 -11469.211} C_VEL
LIN {X 0,Y 390.031,Z 335.524,A -85,B 0,C 180,E1 -11472.372,E2 -11472.372} C_VEL
LIN {X 0,Y 390.043,Z 335.521,A -85,B 0,C 180,E1 -11475.353,E2 -11475.353} C_VEL
LIN {X 0,Y 390.016,Z 335.527,A -85,B 0,C 180,E1 -11478.184,E2 -11478.184} C_VEL
LIN {X 0,Y 390.057,Z 335.522,A -85,B 0,C 180,E1 -11480.903,E2 -11480.903} C_VEL
LIN {X 0,Y 390.083,Z 335.52,A -85,B 0,C 180,E1 -11484.792,E2 -11484.792} C_VEL
LIN {X 0,Y 390.021,Z 335.525,A -85,B 0,C 180,E1 -11488.495,E2 -11488.495} C_VEL
LIN {X 0,Y 390.018,Z 335.524,A -85,B 0,C 180,E1 -11492.003,E2 -11492.003} C_VEL
LIN {X 0,Y 390.045,Z 335.522,A -85,B 0,C 180,E1 -11495.517,E2 -11495.517} C_VEL
LIN {X 0,Y 390.055,Z 335.503,A -85,B 0,C 180,E1 -11498.877,E2 -11498.877} C_VEL
LIN {X 0,Y 390.07,Z 335.514,A -85,B 0,C 180,E1 -11502.164,E2 -11502.164} C_VEL
LIN {X 0,Y 390.095,Z 335.514,A -85,B 0,C 180,E1 -11505.39,E2 -11505.39} C_VEL
LIN {X 0,Y 390.174,Z 335.496,A -85,B 0,C 180,E1 -11507.517,E2 -11507.517} C_VEL
LIN {X 0,Y 390.196,Z 335.494,A -85,B 0,C 180,E1 -11510.671,E2 -11510.671} C_VEL
LIN {X 0,Y 390.287,Z 335.494,A -85,B 0,C 180,E1 -11513.797,E2 -11513.797} C_VEL
LIN {X 0,Y 390.417,Z 335.477,A -85,B 0,C 180,E1 -11517.936,E2 -11517.936} C_VEL
LIN {X 0,Y 390.337,Z 335.479,A -85,B 0,C 180,E1 -11521.031,E2 -11521.031} C_VEL
LIN {X 0,Y 390.264,Z 335.494,A -85,B 0,C 180,E1 -11523.097,E2 -11523.097} C_VEL
LIN {X 0,Y 390.289,Z 335.493,A -85,B 0,C 180,E1 -11526.202,E2 -11526.202} C_VEL
LIN {X 0,Y 390.196,Z 335.502,A -85,B 0,C 180,E1 -11529.329,E2 -11529.329} C_VEL
LIN {X 0,Y 390.173,Z 335.506,A -85,B 0,C 180,E1 -11532.483,E2 -11532.483} C_VEL
LIN {X 0,Y 390.142,Z 335.511,A -85,B 0,C 180,E1 -11535.676,E2 -11535.676} C_VEL
LIN {X 0,Y 390.107,Z 335.512,A -85,B 0,C 180,E1 -11538.922,E2 -11538.922} C_VEL
LIN {X 0,Y 390.042,Z 335.523,A -85,B 0,C 180,E1 -11542.234,E2 -11542.234} C_VEL
LIN {X 0,Y 390.09,Z 335.518,A -85,B 0,C 180,E1 -11545.734,E2 -11545.734} C_VEL
LIN {X 0,Y 390.091,Z 335.519,A -85,B 0,C 180,E1 -11548.017,E2 -11548.017} C_VEL
LIN {X 0,Y 390.026,Z 335.531,A -85,B 0,C 180,E1 -11551.504,E2 -11551.504} C_VEL
LIN {X 0,Y 390.087,Z 335.521,A -85,B 0,C 180,E1 -11555.206,E2 -11555.206} C_VEL
LIN {X 0,Y 390.094,Z 335.517,A -85,B 0,C 180,E1 -11559.092,E2 -11559.092} C_VEL
LIN {X 0,Y 390.044,Z 335.524,A -85,B 0,C 180,E1 -11562.374,E2 -11562.374} C_VEL
LIN {X 0,Y 390.045,Z 335.527,A -85,B 0,C 180,E1 -11565.354,E2 -11565.354} C_VEL
LIN {X 0,Y 390.032,Z 335.525,A -85,B 0,C 180,E1 -11568.186,E2 -11568.186} C_VEL
LIN {X 0,Y 390.092,Z 335.521,A -85,B 0,C 180,E1 -11570.908,E2 -11570.908} C_VEL
LIN {X 0,Y 390.087,Z 335.523,A -85,B 0,C 180,E1 -11574.793,E2 -11574.793} C_VEL
LIN {X 0,Y 390.04,Z 335.526,A -85,B 0,C 180,E1 -11578.497,E2 -11578.497} C_VEL
LIN {X 0,Y 390.101,Z 335.618,A -85,B 0,C 180,E1 -11578.993,E2 -11578.993} C_VEL
LIN {X 0,Y 393.225,Z 349.423,A -85,B 0,C 180,E1 -11582.051,E2 -11582.051} C_VEL
LIN {X 0,Y 394.764,Z 357.94,A -85,B 0,C 180,E1 -11583.856,E2 -11583.856} C_VEL
LIN {X 0,Y 394.037,Z 366.957,A -85,B 0,C 180,E1 -11585.597,E2 -11585.597} C_VEL
LIN {X 0,Y 399.793,Z 400.708,A -85,B 0,C 180,E1 -11586.592,E2 -11586.592} C_VEL
LIN {X 0,Y 398.092,Z 504.408,A -85,B 0,C 180,E1 -11588.477,E2 -11588.477} C_VEL
LIN {X 0,Y 397.483,Z 518.622,A -85,B 0,C 180,E1 -11588.918,E2 -11588.918} C_VEL
LIN {X 0,Y 396.576,Z 532.953,A -85,B 0,C 180,E1 -11589.58,E2 -11589.58} C_VEL
LIN {X 0,Y 395.617,Z 545.985,A -85,B 0,C 180,E1 -11590.394,E2 -11590.394} C_VEL
LIN {X 0,Y 394.502,Z 558.948,A -85,B 0,C 180,E1 -11591.431,E2 -11591.431} C_VEL
LIN {X 0,Y 393.329,Z 570.571,A -85,B 0,C 180,E1 -11592.585,E2 -11592.585} C_VEL
LIN {X 0,Y 392.253,Z 581.228,A -85,B 0,C 180,E1 -11593.876,E2 -11593.876} C_VEL
LIN {X 0,Y 391.161,Z 591.802,A -85,B 0,C 180,E1 -11595.431,E2 -11595.431} C_VEL
LIN {X 0,Y 390.481,Z 600.532,A -85,B 0,C 180,E1 -11596.998,E2 -11596.998} C_VEL
LIN {X 0,Y 389.698,Z 608.882,A -85,B 0,C 180,E1 -11598.821,E2 -11598.821} C_VEL
LIN {X 0,Y 389.171,Z 615.585,A -85,B 0,C 180,E1 -11600.646,E2 -11600.646} C_VEL
LIN {X 0,Y 388.91,Z 621.532,A -85,B 0,C 180,E1 -11602.733,E2 -11602.733} C_VEL
LIN {X 0,Y 388.726,Z 625.88,A -85,B 0,C 180,E1 -11604.814,E2 -11604.814} C_VEL
LIN {X 0,Y 388.631,Z 628.769,A -85,B 0,C 180,E1 -11606.89,E2 -11606.89} C_VEL
LIN {X 0,Y 388.701,Z 630.284,A -85,B 0,C 180,E1 -11608.964,E2 -11608.964} C_VEL
LIN {X 0,Y 388.701,Z 630.456,A -85,B 0,C 180,E1 -11611.036,E2 -11611.036} C_VEL
LIN {X 0,Y 388.628,Z 629.293,A -85,B 0,C 180,E1 -11613.11,E2 -11613.11} C_VEL
LIN {X 0,Y 388.706,Z 626.785,A -85,B 0,C 180,E1 -11615.187,E2 -11615.187} C_VEL
LIN {X 0,Y 388.915,Z 622.848,A -85,B 0,C 180,E1 -11617.267,E2 -11617.267} C_VEL
LIN {X 0,Y 389.262,Z 617.345,A -85,B 0,C 180,E1 -11619.352,E2 -11619.352} C_VEL
LIN {X 0,Y 389.765,Z 611.147,A -85,B 0,C 180,E1 -11621.177,E2 -11621.177} C_VEL
LIN {X 0,Y 390.6,Z 603.435,A -85,B 0,C 180,E1 -11622.998,E2 -11622.998} C_VEL
LIN {X 0,Y 391.443,Z 595.407,A -85,B 0,C 180,E1 -11624.558,E2 -11624.558} C_VEL
LIN {X 0,Y 392.585,Z 585.747,A -85,B 0,C 180,E1 -11626.11,E2 -11626.11} C_VEL
LIN {X 0,Y 393.893,Z 575.048,A -85,B 0,C 180,E1 -11627.523,E2 -11627.523} C_VEL
LIN {X 0,Y 395.283,Z 563.226,A -85,B 0,C 180,E1 -11628.8,E2 -11628.8} C_VEL
LIN {X 0,Y 396.475,Z 551.559,A -85,B 0,C 180,E1 -11629.825,E2 -11629.825} C_VEL
LIN {X 0,Y 397.683,Z 538.069,A -85,B 0,C 180,E1 -11630.766,E2 -11630.766} C_VEL
LIN {X 0,Y 398.685,Z 525.029,A -85,B 0,C 180,E1 -11631.456,E2 -11631.456} C_VEL
LIN {X 0,Y 399.524,Z 511.053,A -85,B 0,C 180,E1 -11631.985,E2 -11631.985} C_VEL
LIN {X 0,Y 400.024,Z 496.442,A -85,B 0,C 180,E1 -11632.329,E2 -11632.329} C_VEL
LIN {X 0,Y 401.748,Z 400.616,A -85,B 0,C 180,E1 -11634.07,E2 -11634.07} C_VEL
LIN {X 0,Y 397.801,Z 379.647,A -85,B 0,C 180,E1 -11634.757,E2 -11634.757} C_VEL
LIN {X 0,Y 395.133,Z 366.75,A -85,B 0,C 180,E1 -11635.23,E2 -11635.23} C_VEL
LIN {X 0,Y 395.707,Z 361.015,A -85,B 0,C 180,E1 -11636.361,E2 -11636.361} C_VEL
LIN {X 0,Y 394.261,Z 352.696,A -85,B 0,C 180,E1 -11638.189,E2 -11638.189} C_VEL
LIN {X 0,Y 391.173,Z 339.985,A -85,B 0,C 180,E1 -11641.153,E2 -11641.153} C_VEL
LIN {X 0,Y 390.038,Z 335.524,A -85,B 0,C 180,E1 -11642.248,E2 -11642.248} C_VEL
LIN {X 0,Y 390.086,Z 335.52,A -85,B 0,C 180,E1 -11645.207,E2 -11645.207} C_VEL
LIN {X 0,Y 390.069,Z 335.516,A -85,B 0,C 180,E1 -11649.218,E2 -11649.218} C_VEL
LIN {X 0,Y 390.044,Z 335.527,A -85,B 0,C 180,E1 -11652.374,E2 -11652.374} C_VEL
LIN {X 0,Y 390.045,Z 335.52,A -85,B 0,C 180,E1 -11655.355,E2 -11655.355} C_VEL
LIN {X 0,Y 390.033,Z 335.523,A -85,B 0,C 180,E1 -11658.187,E2 -11658.187} C_VEL
LIN {X 0,Y 390.093,Z 335.515,A -85,B 0,C 180,E1 -11660.908,E2 -11660.908} C_VEL
LIN {X 0,Y 390.087,Z 335.519,A -85,B 0,C 180,E1 -11664.793,E2 -11664.793} C_VEL
LIN {X 0,Y 390.026,Z 335.528,A -85,B 0,C 180,E1 -11668.496,E2 -11668.496} C_VEL
LIN {X 0,Y 390.041,Z 335.526,A -85,B 0,C 180,E1 -11672.064,E2 -11672.064} C_VEL
LIN {X 0,Y 390.063,Z 335.52,A -85,B 0,C 180,E1 -11675.518,E2 -11675.518} C_VEL
LIN {X 0,Y 390.058,Z 335.519,A -85,B 0,C 180,E1 -11678.878,E2 -11678.878} C_VEL
LIN {X 0,Y 390.131,Z 335.508,A -85,B 0,C 180,E1 -11682.167,E2 -11682.167} C_VEL
LIN {X 0,Y 390.147,Z 335.509,A -85,B 0,C 180,E1 -11685.393,E2 -11685.393} C_VEL
LIN {X 0,Y 390.151,Z 335.51,A -85,B 0,C 180,E1 -11688.572,E2 -11688.572} C_VEL
LIN {X 0,Y 390.26,Z 335.492,A -85,B 0,C 180,E1 -11692.086,E2 -11692.086} C_VEL
LIN {X 0,Y 390.211,Z 335.5,A -85,B 0,C 180,E1 -11694.834,E2 -11694.834} C_VEL
LIN {X 0,Y 390.411,Z 335.475,A -85,B 0,C 180,E1 -11697.937,E2 -11697.937} C_VEL
LIN {X 0,Y 390.293,Z 335.487,A -85,B 0,C 180,E1 -11701.032,E2 -11701.032} C_VEL
LIN {X 0,Y 390.278,Z 335.49,A -85,B 0,C 180,E1 -11703.097,E2 -11703.097} C_VEL
LIN {X 0,Y 390.265,Z 335.486,A -85,B 0,C 180,E1 -11706.455,E2 -11706.455} C_VEL
LIN {X 0,Y 390.196,Z 335.505,A -85,B 0,C 180,E1 -11709.329,E2 -11709.329} C_VEL
LIN {X 0,Y 390.175,Z 335.503,A -85,B 0,C 180,E1 -11712.483,E2 -11712.483} C_VEL
LIN {X 0,Y 390.068,Z 335.517,A -85,B 0,C 180,E1 -11715.68,E2 -11715.68} C_VEL
LIN {X 0,Y 390.051,Z 335.522,A -85,B 0,C 180,E1 -11718.925,E2 -11718.925} C_VEL
LIN {X 0,Y 390.036,Z 335.524,A -85,B 0,C 180,E1 -11722.235,E2 -11722.235} C_VEL
LIN {X 0,Y 390.053,Z 335.522,A -85,B 0,C 180,E1 -11725.722,E2 -11725.722} C_VEL
LIN {X 0,Y 390.025,Z 335.513,A -85,B 0,C 180,E1 -11729.113,E2 -11729.113} C_VEL
LIN {X 0,Y 390.043,Z 335.52,A -85,B 0,C 180,E1 -11732.722,E2 -11732.722} C_VEL
LIN {X 0,Y 390.044,Z 335.508,A -85,B 0,C 180,E1 -11735.822,E2 -11735.822} C_VEL
LIN {X 0,Y 390.037,Z 335.527,A -85,B 0,C 180,E1 -11739.212,E2 -11739.212} C_VEL
LIN {X 0,Y 390.032,Z 335.524,A -85,B 0,C 180,E1 -11742.372,E2 -11742.372} C_VEL
LIN {X 0,Y 390.043,Z 335.518,A -85,B 0,C 180,E1 -11745.354,E2 -11745.354} C_VEL
LIN {X 0,Y 390.017,Z 335.529,A -85,B 0,C 180,E1 -11748.184,E2 -11748.184} C_VEL
LIN {X 0,Y 390.057,Z 335.527,A -85,B 0,C 180,E1 -11750.903,E2 -11750.903} C_VEL
LIN {X 0,Y 390.07,Z 335.524,A -85,B 0,C 180,E1 -11754.791,E2 -11754.791} C_VEL
LIN {X 0,Y 390.107,Z 335.635,A -85,B 0,C 180,E1 -11756.591,E2 -11756.591} C_VEL
LIN {X 0,Y 392.839,Z 347.659,A -85,B 0,C 180,E1 -11759.678,E2 -11759.678} C_VEL
LIN {X 0,Y 399.803,Z 364.38,A -85,B 0,C 180,E1 -11760.524,E2 -11760.524} C_VEL
LIN {X 0,Y 402.224,Z 375.578,A -85,B 0,C 180,E1 -11760.915,E2 -11760.915} C_VEL
LIN {X 0,Y 400.163,Z 483.806,A -85,B 0,C 180,E1 -11762.9,E2 -11762.9} C_VEL
LIN {X 0,Y 399.556,Z 497.898,A -85,B 0,C 180,E1 -11763.35,E2 -11763.35} C_VEL
LIN {X 0,Y 398.649,Z 511.453,A -85,B 0,C 180,E1 -11763.979,E2 -11763.979} C_VEL
LIN {X 0,Y 397.764,Z 523.537,A -85,B 0,C 180,E1 -11764.729,E2 -11764.729} C_VEL
LIN {X 0,Y 396.604,Z 535.595,A -85,B 0,C 180,E1 -11765.669,E2 -11765.669} C_VEL
LIN {X 0,Y 395.276,Z 547.598,A -85,B 0,C 180,E1 -11766.835,E2 -11766.835} C_VEL
LIN {X 0,Y 394.255,Z 557.549,A -85,B 0,C 180,E1 -11768.016,E2 -11768.016} C_VEL
LIN {X 0,Y 393.116,Z 566.843,A -85,B 0,C 180,E1 -11769.324,E2 -11769.324} C_VEL
LIN {X 0,Y 391.959,Z 576.114,A -85,B 0,C 180,E1 -11770.899,E2 -11770.899} C_VEL
LIN {X 0,Y 391.083,Z 583.462,A -85,B 0,C 180,E1 -11772.398,E2 -11772.398} C_VEL
LIN {X 0,Y 390.165,Z 591.129,A -85,B 0,C 180,E1 -11774.324,E2 -11774.324} C_VEL
LIN {X 0,Y 389.534,Z 597.673,A -85,B 0,C 180,E1 -11776.435,E2 -11776.435} C_VEL
LIN {X 0,Y 389.05,Z 602.554,A -85,B 0,C 180,E1 -11778.538,E2 -11778.538} C_VEL
LIN {X 0,Y 388.764,Z 605.925,A -85,B 0,C 180,E1 -11780.636,E2 -11780.636} C_VEL
LIN {X 0,Y 388.678,Z 607.891,A -85,B 0,C 180,E1 -11782.728,E2 -11782.728} C_VEL
LIN {X 0,Y 388.683,Z 608.508,A -85,B 0,C 180,E1 -11784.813,E2 -11784.813} C_VEL
LIN {X 0,Y 388.654,Z 607.803,A -85,B 0,C 180,E1 -11786.89,E2 -11786.89} C_VEL
LIN {X 0,Y 388.749,Z 605.771,A -85,B 0,C 180,E1 -11788.964,E2 -11788.964} C_VEL
LIN {X 0,Y 388.852,Z 602.373,A -85,B 0,C 180,E1 -11791.036,E2 -11791.036} C_VEL
LIN {X 0,Y 389.113,Z 599.091,A -85,B 0,C 180,E1 -11792.506,E2 -11792.506} C_VEL
LIN {X 0,Y 388.723,Z 597.054,A -85,B 0,C 180,E1 -11793.32,E2 -11793.32} C_VEL
LIN {X 0,Y 386.302,Z 593.341,A -85,B 0,C 180,E1 -11794.631,E2 -11794.631} C_VEL
LIN {X 0,Y 383.843,Z 589.02,A -85,B 0,C 180,E1 -11795.916,E2 -11795.916} C_VEL
LIN {X 0,Y 383.406,Z 586.023,A -85,B 0,C 180,E1 -11796.679,E2 -11796.679} C_VEL
LIN {X 0,Y 384.173,Z 578.074,A -85,B 0,C 180,E1 -11798.416,E2 -11798.416} C_VEL
LIN {X 0,Y 384.792,Z 570.963,A -85,B 0,C 180,E1 -11799.727,E2 -11799.727} C_VEL
LIN {X 0,Y 386.07,Z 560.702,A -85,B 0,C 180,E1 -11801.285,E2 -11801.285} C_VEL
LIN {X 0,Y 387.182,Z 549.262,A -85,B 0,C 180,E1 -11802.714,E2 -11802.714} C_VEL
LIN {X 0,Y 388.264,Z 537.844,A -85,B 0,C 180,E1 -11803.877,E2 -11803.877} C_VEL
LIN {X 0,Y 389.346,Z 525.322,A -85,B 0,C 180,E1 -11804.905,E2 -11804.905} C_VEL
LIN {X 0,Y 390.235,Z 512.411,A -85,B 0,C 180,E1 -11805.74,E2 -11805.74} C_VEL
LIN {X 0,Y 391.091,Z 498.49,A -85,B 0,C 180,E1 -11806.408,E2 -11806.408} C_VEL
LIN {X 0,Y 391.619,Z 483.894,A -85,B 0,C 180,E1 -11806.888,E2 -11806.888} C_VEL
LIN {X 0,Y 393.462,Z 374.832,A -85,B 0,C 180,E1 -11808.908,E2 -11808.908} C_VEL
LIN {X 0,Y 390.287,Z 360.386,A -85,B 0,C 180,E1 -11809.381,E2 -11809.381} C_VEL
LIN {X 0,Y 385.402,Z 347.442,A -85,B 0,C 180,E1 -11809.96,E2 -11809.96} C_VEL
LIN {X 0,Y 383.032,Z 336.401,A -85,B 0,C 180,E1 -11812.775,E2 -11812.775} C_VEL
LIN {X 0,Y 382.984,Z 336.407,A -85,B 0,C 180,E1 -11816.131,E2 -11816.131} C_VEL
LIN {X 0,Y 382.976,Z 336.401,A -85,B 0,C 180,E1 -11819.701,E2 -11819.701} C_VEL
LIN {X 0,Y 383.001,Z 336.401,A -85,B 0,C 180,E1 -11823.401,E2 -11823.401} C_VEL
LIN {X 0,Y 383.023,Z 336.398,A -85,B 0,C 180,E1 -11826.162,E2 -11826.162} C_VEL
LIN {X 0,Y 382.986,Z 336.4,A -85,B 0,C 180,E1 -11829.58,E2 -11829.58} C_VEL
LIN {X 0,Y 383.009,Z 336.402,A -85,B 0,C 180,E1 -11832.778,E2 -11832.778} C_VEL
LIN {X 0,Y 382.992,Z 336.398,A -85,B 0,C 180,E1 -11835.788,E2 -11835.788} C_VEL
LIN {X 0,Y 382.963,Z 336.404,A -85,B 0,C 180,E1 -11838.801,E2 -11838.801} C_VEL
LIN {X 0,Y 382.993,Z 336.401,A -85,B 0,C 180,E1 -11842.098,E2 -11842.098} C_VEL
LIN {X 0,Y 383.019,Z 336.397,A -85,B 0,C 180,E1 -11845.332,E2 -11845.332} C_VEL
LIN {X 0,Y 382.982,Z 336.402,A -85,B 0,C 180,E1 -11849.081,E2 -11849.081} C_VEL
LIN {X 0,Y 382.971,Z 336.399,A -85,B 0,C 180,E1 -11852.691,E2 -11852.691} C_VEL
LIN {X 0,Y 383.012,Z 336.402,A -85,B 0,C 180,E1 -11856.191,E2 -11856.191} C_VEL
LIN {X 0,Y 383.044,Z 336.374,A -85,B 0,C 180,E1 -11859.597,E2 -11859.597} C_VEL
LIN {X 0,Y 383.072,Z 336.39,A -85,B 0,C 180,E1 -11862.929,E2 -11862.929} C_VEL
LIN {X 0,Y 383.129,Z 336.377,A -85,B 0,C 180,E1 -11866.464,E2 -11866.464} C_VEL
LIN {X 0,Y 383.146,Z 336.368,A -85,B 0,C 180,E1 -11870.497,E2 -11870.497} C_VEL
LIN {X 0,Y 383.243,Z 336.37,A -85,B 0,C 180,E1 -11873.683,E2 -11873.683} C_VEL
LIN {X 0,Y 383.383,Z 336.353,A -85,B 0,C 180,E1 -11877.899,E2 -11877.899} C_VEL
LIN {X 0,Y 383.377,Z 336.354,A -85,B 0,C 180,E1 -11882.101,E2 -11882.101} C_VEL
LIN {X 0,Y 383.245,Z 336.371,A -85,B 0,C 180,E1 -11886.317,E2 -11886.317} C_VEL
LIN {X 0,Y 383.146,Z 336.382,A -85,B 0,C 180,E1 -11889.502,E2 -11889.502} C_VEL
LIN {X 0,Y 383.128,Z 336.385,A -85,B 0,C 180,E1 -11893.536,E2 -11893.536} C_VEL
LIN {X 0,Y 383.097,Z 336.389,A -85,B 0,C 180,E1 -11897.454,E2 -11897.454} C_VEL
LIN {X 0,Y 383.031,Z 336.395,A -85,B 0,C 180,E1 -11900.647,E2 -11900.647} C_VEL
LIN {X 0,Y 383.03,Z 336.401,A -85,B 0,C 180,E1 -11903.807,E2 -11903.807} C_VEL
LIN {X 0,Y 383.049,Z 336.396,A -85,B 0,C 180,E1 -11907.302,E2 -11907.302} C_VEL
LIN {X 0,Y 382.985,Z 336.404,A -85,B 0,C 180,E1 -11910.918,E2 -11910.918} C_VEL
LIN {X 0,Y 383.02,Z 336.399,A -85,B 0,C 180,E1 -11914.668,E2 -11914.668} C_VEL
LIN {X 0,Y 383.003,Z 336.402,A -85,B 0,C 180,E1 -11917.904,E2 -11917.904} C_VEL
LIN {X 0,Y 382.986,Z 336.407,A -85,B 0,C 180,E1 -11921.347,E2 -11921.347} C_VEL
LIN {X 0,Y 382.997,Z 336.401,A -85,B 0,C 180,E1 -11924.303,E2 -11924.303} C_VEL
LIN {X 0,Y 383.011,Z 336.402,A -85,B 0,C 180,E1 -11927.24,E2 -11927.24} C_VEL
LIN {X 0,Y 383.016,Z 336.401,A -85,B 0,C 180,E1 -11930.413,E2 -11930.413} C_VEL
LIN {X 0,Y 383.028,Z 336.403,A -85,B 0,C 180,E1 -11934.044,E2 -11934.044} C_VEL
LIN {X 0,Y 382.988,Z 336.408,A -85,B 0,C 180,E1 -11937.578,E2 -11937.578} C_VEL
LIN {X 0,Y 383.007,Z 336.456,A -85,B 0,C 180,E1 -11938.623,E2 -11938.623} C_VEL
LIN {X 0,Y 385.965,Z 349.162,A -85,B 0,C 180,E1 -11941.511,E2 -11941.511} C_VEL
LIN {X 0,Y 387.845,Z 358.973,A -85,B 0,C 180,E1 -11943.643,E2 -11943.643} C_VEL
LIN {X 0,Y 387.244,Z 366.783,A -85,B 0,C 180,E1 -11945.185,E2 -11945.185} C_VEL
LIN {X 0,Y 393.191,Z 401.938,A -85,B 0,C 180,E1 -11946.239,E2 -11946.239} C_VEL
LIN {X 0,Y 391.434,Z 504.192,A -85,B 0,C 180,E1 -11948.127,E2 -11948.127} C_VEL
LIN {X 0,Y 390.796,Z 518.413,A -85,B 0,C 180,E1 -11948.574,E2 -11948.574} C_VEL
LIN {X 0,Y 389.917,Z 532.176,A -85,B 0,C 180,E1 -11949.215,E2 -11949.215} C_VEL
LIN {X 0,Y 388.894,Z 544.887,A -85,B 0,C 180,E1 -11950.006,E2 -11950.006} C_VEL
LIN {X 0,Y 387.886,Z 556.951,A -85,B 0,C 180,E1 -11950.965,E2 -11950.965} C_VEL
LIN {X 0,Y 386.641,Z 568.891,A -85,B 0,C 180,E1 -11952.137,E2 -11952.137} C_VEL
LIN {X 0,Y 385.382,Z 580.782,A -85,B 0,C 180,E1 -11953.581,E2 -11953.581} C_VEL
LIN {X 0,Y 384.214,Z 591.396,A -85,B 0,C 180,E1 -11955.162,E2 -11955.162} C_VEL
LIN {X 0,Y 383.519,Z 600.162,A -85,B 0,C 180,E1 -11956.758,E2 -11956.758} C_VEL
LIN {X 0,Y 382.683,Z 608.551,A -85,B 0,C 180,E1 -11958.614,E2 -11958.614} C_VEL
LIN {X 0,Y 382.11,Z 615.283,A -85,B 0,C 180,E1 -11960.472,E2 -11960.472} C_VEL
LIN {X 0,Y 381.827,Z 621.254,A -85,B 0,C 180,E1 -11962.597,E2 -11962.597} C_VEL
LIN {X 0,Y 381.634,Z 625.624,A -85,B 0,C 180,E1 -11964.717,E2 -11964.717} C_VEL
LIN {X 0,Y 381.542,Z 628.534,A -85,B 0,C 180,E1 -11966.832,E2 -11966.832} C_VEL
LIN {X 0,Y 381.616,Z 630.069,A -85,B 0,C 180,E1 -11968.945,E2 -11968.945} C_VEL
LIN {X 0,Y 381.615,Z 630.259,A -85,B 0,C 180,E1 -11971.055,E2 -11971.055} C_VEL
LIN {X 0,Y 381.539,Z 629.115,A -85,B 0,C 180,E1 -11973.168,E2 -11973.168} C_VEL
LIN {X 0,Y 381.616,Z 626.626,A -85,B 0,C 180,E1 -11975.283,E2 -11975.283} C_VEL
LIN {X 0,Y 381.837,Z 622.718,A -85,B 0,C 180,E1 -11977.403,E2 -11977.403} C_VEL
LIN {X 0,Y 382.198,Z 617.24,A -85,B 0,C 180,E1 -11979.526,E2 -11979.526} C_VEL
LIN {X 0,Y 382.776,Z 611.068,A -85,B 0,C 180,E1 -11981.384,E2 -11981.384} C_VEL
LIN {X 0,Y 383.609,Z 603.384,A -85,B 0,C 180,E1 -11983.239,E2 -11983.239} C_VEL
LIN {X 0,Y 384.716,Z 593.902,A -85,B 0,C 180,E1 -11985.089,E2 -11985.089} C_VEL
LIN {X 0,Y 385.939,Z 583.986,A -85,B 0,C 180,E1 -11986.667,E2 -11986.667} C_VEL
LIN {X 0,Y 387.413,Z 572.979,A -85,B 0,C 180,E1 -11988.099,E2 -11988.099} C_VEL
LIN {X 0,Y 388.88,Z 560.726,A -85,B 0,C 180,E1 -11989.395,E2 -11989.395} C_VEL
LIN {X 0,Y 390.177,Z 548.354,A -85,B 0,C 180,E1 -11990.445,E2 -11990.445} C_VEL
LIN {X 0,Y 391.308,Z 535.174,A -85,B 0,C 180,E1 -11991.328,E2 -11991.328} C_VEL
LIN {X 0,Y 392.418,Z 521.15,A -85,B 0,C 180,E1 -11992.023,E2 -11992.023} C_VEL
LIN {X 0,Y 393.262,Z 506.35,A -85,B 0,C 180,E1 -11992.527,E2 -11992.527} C_VEL
LIN {X 0,Y 393.93,Z 478.537,A -85,B 0,C 180,E1 -11993.075,E2 -11993.075} C_VEL
LIN {X 0,Y 395.304,Z 401.234,A -85,B 0,C 180,E1 -11994.508,E2 -11994.508} C_VEL
LIN {X 0,Y 391.405,Z 380.744,A -85,B 0,C 180,E1 -11995.201,E2 -11995.201} C_VEL
LIN {X 0,Y 388.452,Z 366.541,A -85,B 0,C 180,E1 -11995.736,E2 -11995.736} C_VEL
LIN {X 0,Y 388.846,Z 362.387,A -85,B 0,C 180,E1 -11996.573,E2 -11996.573} C_VEL
LIN {X 0,Y 387.364,Z 354.204,A -85,B 0,C 180,E1 -11998.415,E2 -11998.415} C_VEL
LIN {X 0,Y 384.345,Z 341.628,A -85,B 0,C 180,E1 -12001.408,E2 -12001.408} C_VEL
LIN {X 0,Y 383.018,Z 336.399,A -85,B 0,C 180,E1 -12002.729,E2 -12002.729} C_VEL
LIN {X 0,Y 383.033,Z 336.398,A -85,B 0,C 180,E1 -12006.165,E2 -12006.165} C_VEL
LIN {X 0,Y 383.009,Z 336.399,A -85,B 0,C 180,E1 -12009.959,E2 -12009.959} C_VEL
LIN {X 0,Y 383.006,Z 336.4,A -85,B 0,C 180,E1 -12012.779,E2 -12012.779} C_VEL
LIN {X 0,Y 382.998,Z 336.398,A -85,B 0,C 180,E1 -12015.79,E2 -12015.79} C_VEL
LIN {X 0,Y 382.991,Z 336.403,A -85,B 0,C 180,E1 -12018.796,E2 -12018.796} C_VEL
LIN {X 0,Y 383.002,Z 336.401,A -85,B 0,C 180,E1 -12022.097,E2 -12022.097} C_VEL
LIN {X 0,Y 383.02,Z 336.397,A -85,B 0,C 180,E1 -12025.332,E2 -12025.332} C_VEL
LIN {X 0,Y 382.984,Z 336.401,A -85,B 0,C 180,E1 -12029.082,E2 -12029.082} C_VEL
LIN {X 0,Y 382.996,Z 336.399,A -85,B 0,C 180,E1 -12032.694,E2 -12032.694} C_VEL
LIN {X 0,Y 383.019,Z 336.401,A -85,B 0,C 180,E1 -12036.192,E2 -12036.192} C_VEL
LIN {X 0,Y 383.058,Z 336.392,A -85,B 0,C 180,E1 -12039.599,E2 -12039.599} C_VEL
LIN {X 0,Y 383.108,Z 336.383,A -85,B 0,C 180,E1 -12042.932,E2 -12042.932} C_VEL
LIN {X 0,Y 383.129,Z 336.377,A -85,B 0,C 180,E1 -12046.464,E2 -12046.464} C_VEL
LIN {X 0,Y 383.134,Z 336.384,A -85,B 0,C 180,E1 -12049.43,E2 -12049.43} C_VEL
LIN {X 0,Y 383.204,Z 336.373,A -85,B 0,C 180,E1 -12052.624,E2 -12052.624} C_VEL
LIN {X 0,Y 383.182,Z 336.376,A -85,B 0,C 180,E1 -12054.739,E2 -12054.739} C_VEL
LIN {X 0,Y 383.377,Z 336.351,A -85,B 0,C 180,E1 -12057.899,E2 -12057.899} C_VEL
LIN {X 0,Y 383.383,Z 336.347,A -85,B 0,C 180,E1 -12062.101,E2 -12062.101} C_VEL
LIN {X 0,Y 383.231,Z 336.362,A -85,B 0,C 180,E1 -12066.442,E2 -12066.442} C_VEL
LIN {X 0,Y 383.146,Z 336.385,A -85,B 0,C 180,E1 -12069.503,E2 -12069.503} C_VEL
LIN {X 0,Y 383.13,Z 336.385,A -85,B 0,C 180,E1 -12073.536,E2 -12073.536} C_VEL
LIN {X 0,Y 383.029,Z 336.393,A -85,B 0,C 180,E1 -12077.421,E2 -12077.421} C_VEL
LIN {X 0,Y 383.017,Z 336.391,A -85,B 0,C 180,E1 -12080.641,E2 -12080.641} C_VEL
LIN {X 0,Y 383.011,Z 336.397,A -85,B 0,C 180,E1 -12083.809,E2 -12083.809} C_VEL
LIN {X 0,Y 382.971,Z 336.407,A -85,B 0,C 180,E1 -12087.309,E2 -12087.309} C_VEL
LIN {X 0,Y 382.982,Z 336.381,A -85,B 0,C 180,E1 -12090.919,E2 -12090.919} C_VEL
LIN {X 0,Y 383.014,Z 336.397,A -85,B 0,C 180,E1 -12094.669,E2 -12094.669} C_VEL
LIN {X 0,Y 382.993,Z 336.397,A -85,B 0,C 180,E1 -12097.902,E2 -12097.902} C_VEL
LIN {X 0,Y 382.963,Z 336.408,A -85,B 0,C 180,E1 -12101.351,E2 -12101.351} C_VEL
LIN {X 0,Y 382.991,Z 336.403,A -85,B 0,C 180,E1 -12104.302,E2 -12104.302} C_VEL
LIN {X 0,Y 382.985,Z 336.405,A -85,B 0,C 180,E1 -12107.236,E2 -12107.236} C_VEL
LIN {X 0,Y 382.986,Z 336.405,A -85,B 0,C 180,E1 -12110.42,E2 -12110.42} C_VEL
LIN {X 0,Y 383.015,Z 336.401,A -85,B 0,C 180,E1 -12114.043,E2 -12114.043} C_VEL
LIN {X 0,Y 383.06,Z 336.525,A -85,B 0,C 180,E1 -12116.141,E2 -12116.141} C_VEL
LIN {X 0,Y 385.614,Z 347.746,A -85,B 0,C 180,E1 -12119.121,E2 -12119.121} C_VEL
LIN {X 0,Y 393.632,Z 366.529,A -85,B 0,C 180,E1 -12120.117,E2 -12120.117} C_VEL
LIN {X 0,Y 395.807,Z 375.974,A -85,B 0,C 180,E1 -12120.465,E2 -12120.465} C_VEL
LIN {X 0,Y 393.704,Z 484.3,A -85,B 0,C 180,E1 -12122.49,E2 -12122.49} C_VEL
LIN {X 0,Y 393.041,Z 499.054,A -85,B 0,C 180,E1 -12122.98,E2 -12122.98} C_VEL
LIN {X 0,Y 392.084,Z 512.166,A -85,B 0,C 180,E1 -12123.606,E2 -12123.606} C_VEL
LIN {X 0,Y 391.232,Z 523.251,A -85,B 0,C 180,E1 -12124.301,E2 -12124.301} C_VEL
LIN {X 0,Y 390.062,Z 535.157,A -85,B 0,C 180,E1 -12125.234,E2 -12125.234} C_VEL
LIN {X 0,Y 388.664,Z 547.271,A -85,B 0,C 180,E1 -12126.417,E2 -12126.417} C_VEL
LIN {X 0,Y 387.554,Z 557.53,A -85,B 0,C 180,E1 -12127.647,E2 -12127.647} C_VEL
LIN {X 0,Y 386.149,Z 568.317,A -85,B 0,C 180,E1 -12129.212,E2 -12129.212} C_VEL
LIN {X 0,Y 384.949,Z 577.372,A -85,B 0,C 180,E1 -12130.814,E2 -12130.814} C_VEL
LIN {X 0,Y 383.987,Z 585.101,A -85,B 0,C 180,E1 -12132.475,E2 -12132.475} C_VEL
LIN {X 0,Y 383.216,Z 591.127,A -85,B 0,C 180,E1 -12134.032,E2 -12134.032} C_VEL
LIN {X 0,Y 382.525,Z 597.715,A -85,B 0,C 180,E1 -12136.182,E2 -12136.182} C_VEL
LIN {X 0,Y 381.988,Z 602.637,A -85,B 0,C 180,E1 -12138.324,E2 -12138.324} C_VEL
LIN {X 0,Y 381.69,Z 606.045,A -85,B 0,C 180,E1 -12140.461,E2 -12140.461} C_VEL
LIN {X 0,Y 381.591,Z 608.051,A -85,B 0,C 180,E1 -12142.593,E2 -12142.593} C_VEL
LIN {X 0,Y 381.592,Z 608.712,A -85,B 0,C 180,E1 -12144.716,E2 -12144.716} C_VEL
LIN {X 0,Y 381.562,Z 608.049,A -85,B 0,C 180,E1 -12146.832,E2 -12146.832} C_VEL
LIN {X 0,Y 381.68,Z 606.053,A -85,B 0,C 180,E1 -12148.945,E2 -12148.945} C_VEL
LIN {X 0,Y 381.781,Z 602.693,A -85,B 0,C 180,E1 -12151.055,E2 -12151.055} C_VEL
LIN {X 0,Y 382.166,Z 597.861,A -85,B 0,C 180,E1 -12153.163,E2 -12153.163} C_VEL
LIN {X 0,Y 382.701,Z 593.198,A -85,B 0,C 180,E1 -12154.74,E2 -12154.74} C_VEL
LIN {X 0,Y 383.406,Z 586.023,A -85,B 0,C 180,E1 -12156.679,E2 -12156.679} C_VEL
LIN {X 0,Y 383,Z 582.931,A -85,B 0,C 180,E1 -12157.425,E2 -12157.425} C_VEL
LIN {X 0,Y 380.713,Z 577.617,A -85,B 0,C 180,E1 -12158.634,E2 -12158.634} C_VEL
LIN {X 0,Y 378.54,Z 571.9,A -85,B 0,C 180,E1 -12159.807,E2 -12159.807} C_VEL
LIN {X 0,Y 378.312,Z 568.009,A -85,B 0,C 180,E1 -12160.484,E2 -12160.484} C_VEL
LIN {X 0,Y 379.572,Z 557.471,A -85,B 0,C 180,E1 -12162.023,E2 -12162.023} C_VEL
LIN {X 0,Y 380.684,Z 546.489,A -85,B 0,C 180,E1 -12163.342,E2 -12163.342} C_VEL
LIN {X 0,Y 381.805,Z 534.398,A -85,B 0,C 180,E1 -12164.525,E2 -12164.525} C_VEL
LIN {X 0,Y 382.962,Z 520.838,A -85,B 0,C 180,E1 -12165.569,E2 -12165.569} C_VEL
LIN {X 0,Y 383.917,Z 507.657,A -85,B 0,C 180,E1 -12166.347,E2 -12166.347} C_VEL
LIN {X 0,Y 384.63,Z 493.335,A -85,B 0,C 180,E1 -12166.965,E2 -12166.965} C_VEL
LIN {X 0,Y 385.107,Z 479.336,A -85,B 0,C 180,E1 -12167.353,E2 -12167.353} C_VEL
LIN {X 0,Y 386.959,Z 376.612,A -85,B 0,C 180,E1 -12169.267,E2 -12169.267} C_VEL
LIN {X 0,Y 384.084,Z 362.987,A -85,B 0,C 180,E1 -12169.716,E2 -12169.716} C_VEL
LIN {X 0,Y 378.209,Z 347.65,A -85,B 0,C 180,E1 -12170.424,E2 -12170.424} C_VEL
LIN {X 0,Y 376.001,Z 337.276,A -85,B 0,C 180,E1 -12173.112,E2 -12173.112} C_VEL
LIN {X 0,Y 375.912,Z 337.289,A -85,B 0,C 180,E1 -12176.66,E2 -12176.66} C_VEL
LIN {X 0,Y 375.915,Z 337.285,A -85,B 0,C 180,E1 -12179.084,E2 -12179.084} C_VEL
LIN {X 0,Y 375.938,Z 337.281,A -85,B 0,C 180,E1 -12181.564,E2 -12181.564} C_VEL
LIN {X 0,Y 375.977,Z 337.277,A -85,B 0,C 180,E1 -12184.666,E2 -12184.666} C_VEL
LIN {X 0,Y 375.935,Z 337.282,A -85,B 0,C 180,E1 -12188.262,E2 -12188.262} C_VEL
LIN {X 0,Y 375.915,Z 337.28,A -85,B 0,C 180,E1 -12191.597,E2 -12191.597} C_VEL
LIN {X 0,Y 375.923,Z 337.281,A -85,B 0,C 180,E1 -12194.73,E2 -12194.73} C_VEL
LIN {X 0,Y 375.91,Z 337.282,A -85,B 0,C 180,E1 -12197.696,E2 -12197.696} C_VEL
LIN {X 0,Y 375.935,Z 337.284,A -85,B 0,C 180,E1 -12200.533,E2 -12200.533} C_VEL
LIN {X 0,Y 375.963,Z 337.273,A -85,B 0,C 180,E1 -12203.496,E2 -12203.496} C_VEL
LIN {X 0,Y 375.962,Z 337.277,A -85,B 0,C 180,E1 -12205.888,E2 -12205.888} C_VEL
LIN {X 0,Y 375.962,Z 337.276,A -85,B 0,C 180,E1 -12209.687,E2 -12209.687} C_VEL
LIN {X 0,Y 375.92,Z 337.278,A -85,B 0,C 180,E1 -12212.135,E2 -12212.135} C_VEL
LIN {X 0,Y 375.939,Z 337.283,A -85,B 0,C 180,E1 -12214.534,E2 -12214.534} C_VEL
LIN {X 0,Y 375.977,Z 337.271,A -85,B 0,C 180,E1 -12216.887,E2 -12216.887} C_VEL
LIN {X 0,Y 375.978,Z 337.256,A -85,B 0,C 180,E1 -12220.338,E2 -12220.338} C_VEL
LIN {X 0,Y 375.977,Z 337.274,A -85,B 0,C 180,E1 -12223.716,E2 -12223.716} C_VEL
LIN {X 0,Y 376.107,Z 337.247,A -85,B 0,C 180,E1 -12227.042,E2 -12227.042} C_VEL
LIN {X 0,Y 376.116,Z 337.24,A -85,B 0,C 180,E1 -12230.318,E2 -12230.318} C_VEL
LIN {X 0,Y 376.202,Z 337.246,A -85,B 0,C 180,E1 -12233.564,E2 -12233.564} C_VEL
LIN {X 0,Y 376.348,Z 337.229,A -85,B 0,C 180,E1 -12237.859,E2 -12237.859} C_VEL
LIN {X 0,Y 376.342,Z 337.231,A -85,B 0,C 180,E1 -12242.14,E2 -12242.14} C_VEL
LIN {X 0,Y 376.203,Z 337.247,A -85,B 0,C 180,E1 -12246.435,E2 -12246.435} C_VEL
LIN {X 0,Y 376.116,Z 337.258,A -85,B 0,C 180,E1 -12249.681,E2 -12249.681} C_VEL
LIN {X 0,Y 376.092,Z 337.262,A -85,B 0,C 180,E1 -12253.657,E2 -12253.657} C_VEL
LIN {X 0,Y 376.046,Z 337.269,A -85,B 0,C 180,E1 -12257.607,E2 -12257.607} C_VEL
LIN {X 0,Y 375.98,Z 337.274,A -85,B 0,C 180,E1 -12260.832,E2 -12260.832} C_VEL
LIN {X 0,Y 375.985,Z 337.275,A -85,B 0,C 180,E1 -12264.282,E2 -12264.282} C_VEL
LIN {X 0,Y 375.979,Z 337.279,A -85,B 0,C 180,E1 -12267.86,E2 -12267.86} C_VEL
LIN {X 0,Y 375.96,Z 337.283,A -85,B 0,C 180,E1 -12271.562,E2 -12271.562} C_VEL
LIN {X 0,Y 375.96,Z 337.281,A -85,B 0,C 180,E1 -12275.415,E2 -12275.415} C_VEL
LIN {X 0,Y 375.978,Z 337.275,A -85,B 0,C 180,E1 -12278.271,E2 -12278.271} C_VEL
LIN {X 0,Y 375.936,Z 337.286,A -85,B 0,C 180,E1 -12281.601,E2 -12281.601} C_VEL
LIN {X 0,Y 375.928,Z 337.286,A -85,B 0,C 180,E1 -12285.268,E2 -12285.268} C_VEL
LIN {X 0,Y 375.935,Z 337.281,A -85,B 0,C 180,E1 -12288.399,E2 -12288.399} C_VEL
LIN {X 0,Y 375.976,Z 337.281,A -85,B 0,C 180,E1 -12291.729,E2 -12291.729} C_VEL
LIN {X 0,Y 375.981,Z 337.283,A -85,B 0,C 180,E1 -12295.332,E2 -12295.332} C_VEL
LIN {X 0,Y 375.985,Z 337.468,A -85,B 0,C 180,E1 -12298.283,E2 -12298.283} C_VEL
LIN {X 0,Y 379.201,Z 351.316,A -85,B 0,C 180,E1 -12301.494,E2 -12301.494} C_VEL
LIN {X 0,Y 380.89,Z 359.992,A -85,B 0,C 180,E1 -12303.42,E2 -12303.42} C_VEL
LIN {X 0,Y 380.5,Z 366.896,A -85,B 0,C 180,E1 -12304.772,E2 -12304.772} C_VEL
LIN {X 0,Y 386.596,Z 402.482,A -85,B 0,C 180,E1 -12305.859,E2 -12305.859} C_VEL
LIN {X 0,Y 384.786,Z 503.953,A -85,B 0,C 180,E1 -12307.764,E2 -12307.764} C_VEL
LIN {X 0,Y 384.121,Z 518.193,A -85,B 0,C 180,E1 -12308.218,E2 -12308.218} C_VEL
LIN {X 0,Y 383.148,Z 532.528,A -85,B 0,C 180,E1 -12308.901,E2 -12308.901} C_VEL
LIN {X 0,Y 382.073,Z 545.538,A -85,B 0,C 180,E1 -12309.737,E2 -12309.737} C_VEL
LIN {X 0,Y 380.981,Z 557.82,A -85,B 0,C 180,E1 -12310.747,E2 -12310.747} C_VEL
LIN {X 0,Y 379.713,Z 569.573,A -85,B 0,C 180,E1 -12311.939,E2 -12311.939} C_VEL
LIN {X 0,Y 378.499,Z 580.329,A -85,B 0,C 180,E1 -12313.273,E2 -12313.273} C_VEL
LIN {X 0,Y 377.308,Z 590.987,A -85,B 0,C 180,E1 -12314.884,E2 -12314.884} C_VEL
LIN {X 0,Y 376.534,Z 599.921,A -85,B 0,C 180,E1 -12316.535,E2 -12316.535} C_VEL
LIN {X 0,Y 375.678,Z 608.213,A -85,B 0,C 180,E1 -12318.398,E2 -12318.398} C_VEL
LIN {X 0,Y 375.067,Z 614.977,A -85,B 0,C 180,E1 -12320.291,E2 -12320.291} C_VEL
LIN {X 0,Y 374.729,Z 620.974,A -85,B 0,C 180,E1 -12322.456,E2 -12322.456} C_VEL
LIN {X 0,Y 374.546,Z 625.367,A -85,B 0,C 180,E1 -12324.617,E2 -12324.617} C_VEL
LIN {X 0,Y 374.539,Z 627.01,A -85,B 0,C 180,E1 -12325.695,E2 -12325.695} C_VEL
LIN {X 0,Y 374.471,Z 629.244,A -85,B 0,C 180,E1 -12327.849,E2 -12327.849} C_VEL
LIN {X 0,Y 374.552,Z 630.125,A -85,B 0,C 180,E1 -12330,E2 -12330} C_VEL
LIN {X 0,Y 374.455,Z 629.666,A -85,B 0,C 180,E1 -12332.151,E2 -12332.151} C_VEL
LIN {X 0,Y 374.513,Z 627.875,A -85,B 0,C 180,E1 -12334.305,E2 -12334.305} C_VEL
LIN {X 0,Y 374.629,Z 624.712,A -85,B 0,C 180,E1 -12336.463,E2 -12336.463} C_VEL
LIN {X 0,Y 374.917,Z 620.067,A -85,B 0,C 180,E1 -12338.625,E2 -12338.625} C_VEL
LIN {X 0,Y 375.429,Z 613.785,A -85,B 0,C 180,E1 -12340.789,E2 -12340.789} C_VEL
LIN {X 0,Y 376.345,Z 606.81,A -85,B 0,C 180,E1 -12342.675,E2 -12342.675} C_VEL
LIN {X 0,Y 377.253,Z 598.183,A -85,B 0,C 180,E1 -12344.566,E2 -12344.566} C_VEL
LIN {X 0,Y 378.457,Z 589.182,A -85,B 0,C 180,E1 -12346.174,E2 -12346.174} C_VEL
LIN {X 0,Y 379.936,Z 578.304,A -85,B 0,C 180,E1 -12347.771,E2 -12347.771} C_VEL
LIN {X 0,Y 381.411,Z 567.281,A -85,B 0,C 180,E1 -12349.091,E2 -12349.091} C_VEL
LIN {X 0,Y 382.851,Z 555.19,A -85,B 0,C 180,E1 -12350.273,E2 -12350.273} C_VEL
LIN {X 0,Y 384.021,Z 543.3,A -85,B 0,C 180,E1 -12351.211,E2 -12351.211} C_VEL
LIN {X 0,Y 385.222,Z 529.841,A -85,B 0,C 180,E1 -12352.033,E2 -12352.033} C_VEL
LIN {X 0,Y 386.301,Z 515.301,A -85,B 0,C 180,E1 -12352.673,E2 -12352.673} C_VEL
LIN {X 0,Y 387.02,Z 500.859,A -85,B 0,C 180,E1 -12353.087,E2 -12353.087} C_VEL
LIN {X 0,Y 388.949,Z 402.325,A -85,B 0,C 180,E1 -12354.947,E2 -12354.947} C_VEL
LIN {X 0,Y 383.827,Z 375.624,A -85,B 0,C 180,E1 -12355.882,E2 -12355.882} C_VEL
LIN {X 0,Y 381.807,Z 366.35,A -85,B 0,C 180,E1 -12356.254,E2 -12356.254} C_VEL
LIN {X 0,Y 381.829,Z 362.376,A -85,B 0,C 180,E1 -12357.101,E2 -12357.101} C_VEL
LIN {X 0,Y 379.516,Z 351.45,A -85,B 0,C 180,E1 -12359.663,E2 -12359.663} C_VEL
LIN {X 0,Y 376.341,Z 338.745,A -85,B 0,C 180,E1 -12362.822,E2 -12362.822} C_VEL
LIN {X 0,Y 375.983,Z 337.275,A -85,B 0,C 180,E1 -12363.224,E2 -12363.224} C_VEL
LIN {X 0,Y 375.954,Z 337.281,A -85,B 0,C 180,E1 -12366.741,E2 -12366.741} C_VEL
LIN {X 0,Y 375.989,Z 337.274,A -85,B 0,C 180,E1 -12369.971,E2 -12369.971} C_VEL
LIN {X 0,Y 375.93,Z 337.278,A -85,B 0,C 180,E1 -12373.766,E2 -12373.766} C_VEL
LIN {X 0,Y 375.936,Z 337.282,A -85,B 0,C 180,E1 -12376.811,E2 -12376.811} C_VEL
LIN {X 0,Y 375.965,Z 337.275,A -85,B 0,C 180,E1 -12380.538,E2 -12380.538} C_VEL
LIN {X 0,Y 375.965,Z 337.273,A -85,B 0,C 180,E1 -12383.496,E2 -12383.496} C_VEL
LIN {X 0,Y 375.962,Z 337.279,A -85,B 0,C 180,E1 -12385.889,E2 -12385.889} C_VEL
LIN {X 0,Y 375.964,Z 337.276,A -85,B 0,C 180,E1 -12389.688,E2 -12389.688} C_VEL
LIN {X 0,Y 375.942,Z 337.276,A -85,B 0,C 180,E1 -12393.342,E2 -12393.342} C_VEL
LIN {X 0,Y 375.98,Z 337.271,A -85,B 0,C 180,E1 -12396.887,E2 -12396.887} C_VEL
LIN {X 0,Y 376.001,Z 337.274,A -85,B 0,C 180,E1 -12400.34,E2 -12400.34} C_VEL
LIN {X 0,Y 376.032,Z 337.267,A -85,B 0,C 180,E1 -12403.719,E2 -12403.719} C_VEL
LIN {X 0,Y 376.107,Z 337.25,A -85,B 0,C 180,E1 -12407.042,E2 -12407.042} C_VEL
LIN {X 0,Y 376.116,Z 337.255,A -85,B 0,C 180,E1 -12410.319,E2 -12410.319} C_VEL
LIN {X 0,Y 376.204,Z 337.246,A -85,B 0,C 180,E1 -12413.565,E2 -12413.565} C_VEL
LIN {X 0,Y 376.342,Z 337.226,A -85,B 0,C 180,E1 -12417.86,E2 -12417.86} C_VEL
LIN {X 0,Y 376.348,Z 337.224,A -85,B 0,C 180,E1 -12422.141,E2 -12422.141} C_VEL
LIN {X 0,Y 376.201,Z 337.237,A -85,B 0,C 180,E1 -12426.436,E2 -12426.436} C_VEL
LIN {X 0,Y 376.116,Z 337.262,A -85,B 0,C 180,E1 -12429.682,E2 -12429.682} C_VEL
LIN {X 0,Y 376.094,Z 337.263,A -85,B 0,C 180,E1 -12433.658,E2 -12433.658} C_VEL
LIN {X 0,Y 375.987,Z 337.272,A -85,B 0,C 180,E1 -12437.578,E2 -12437.578} C_VEL
LIN {X 0,Y 375.982,Z 337.267,A -85,B 0,C 180,E1 -12440.832,E2 -12440.832} C_VEL
LIN {X 0,Y 375.938,Z 337.275,A -85,B 0,C 180,E1 -12444.286,E2 -12444.286} C_VEL
LIN {X 0,Y 375.914,Z 337.283,A -85,B 0,C 180,E1 -12446.661,E2 -12446.661} C_VEL
LIN {X 0,Y 375.915,Z 337.27,A -85,B 0,C 180,E1 -12449.084,E2 -12449.084} C_VEL
LIN {X 0,Y 375.94,Z 337.265,A -85,B 0,C 180,E1 -12451.564,E2 -12451.564} C_VEL
LIN {X 0,Y 375.978,Z 337.274,A -85,B 0,C 180,E1 -12454.666,E2 -12454.666} C_VEL
LIN {X 0,Y 375.935,Z 337.279,A -85,B 0,C 180,E1 -12458.262,E2 -12458.262} C_VEL
LIN {X 0,Y 375.916,Z 337.286,A -85,B 0,C 180,E1 -12461.597,E2 -12461.597} C_VEL
LIN {X 0,Y 375.923,Z 337.283,A -85,B 0,C 180,E1 -12464.73,E2 -12464.73} C_VEL
LIN {X 0,Y 375.91,Z 337.289,A -85,B 0,C 180,E1 -12467.696,E2 -12467.696} C_VEL
LIN {X 0,Y 375.935,Z 337.284,A -85,B 0,C 180,E1 -12470.534,E2 -12470.534} C_VEL
LIN {X 0,Y 375.959,Z 337.282,A -85,B 0,C 180,E1 -12473.497,E2 -12473.497} C_VEL
LIN {X 0,Y 376.006,Z 337.477,A -85,B 0,C 180,E1 -12475.685,E2 -12475.685} C_VEL
LIN {X 0,Y 378.503,Z 348.045,A -85,B 0,C 180,E1 -12478.552,E2 -12478.552} C_VEL
LIN {X 0,Y 387.614,Z 369.101,A -85,B 0,C 180,E1 -12479.716,E2 -12479.716} C_VEL
LIN {X 0,Y 389.488,Z 377.768,A -85,B 0,C 180,E1 -12480.035,E2 -12480.035} C_VEL
LIN {X 0,Y 387.265,Z 484.794,A -85,B 0,C 180,E1 -12482.067,E2 -12482.067} C_VEL
LIN {X 0,Y 386.564,Z 499.446,A -85,B 0,C 180,E1 -12482.563,E2 -12482.563} C_VEL
LIN {X 0,Y 385.492,Z 513.325,A -85,B 0,C 180,E1 -12483.244,E2 -12483.244} C_VEL
LIN {X 0,Y 384.412,Z 526.449,A -85,B 0,C 180,E1 -12484.119,E2 -12484.119} C_VEL
LIN {X 0,Y 383.01,Z 539.039,A -85,B 0,C 180,E1 -12485.181,E2 -12485.181} C_VEL
LIN {X 0,Y 381.646,Z 550.504,A -85,B 0,C 180,E1 -12486.389,E2 -12486.389} C_VEL
LIN {X 0,Y 380.291,Z 561.89,A -85,B 0,C 180,E1 -12487.865,E2 -12487.865} C_VEL
LIN {X 0,Y 378.953,Z 571.424,A -85,B 0,C 180,E1 -12489.367,E2 -12489.367} C_VEL
LIN {X 0,Y 377.771,Z 579.985,A -85,B 0,C 180,E1 -12491,E2 -12491} C_VEL
LIN {X 0,Y 376.708,Z 588.128,A -85,B 0,C 180,E1 -12492.912,E2 -12492.912} C_VEL
LIN {X 0,Y 375.863,Z 594.663,A -85,B 0,C 180,E1 -12494.824,E2 -12494.824} C_VEL
LIN {X 0,Y 375.202,Z 600.221,A -85,B 0,C 180,E1 -12496.914,E2 -12496.914} C_VEL
LIN {X 0,Y 374.75,Z 604.625,A -85,B 0,C 180,E1 -12499.191,E2 -12499.191} C_VEL
LIN {X 0,Y 374.534,Z 607.358,A -85,B 0,C 180,E1 -12501.366,E2 -12501.366} C_VEL
LIN {X 0,Y 374.535,Z 608.723,A -85,B 0,C 180,E1 -12503.535,E2 -12503.535} C_VEL
LIN {X 0,Y 374.518,Z 608.764,A -85,B 0,C 180,E1 -12505.695,E2 -12505.695} C_VEL
LIN {X 0,Y 374.531,Z 607.481,A -85,B 0,C 180,E1 -12507.849,E2 -12507.849} C_VEL
LIN {X 0,Y 374.626,Z 604.85,A -85,B 0,C 180,E1 -12510,E2 -12510} C_VEL
LIN {X 0,Y 374.853,Z 600.809,A -85,B 0,C 180,E1 -12512.149,E2 -12512.149} C_VEL
LIN {X 0,Y 375.448,Z 595.226,A -85,B 0,C 180,E1 -12514.294,E2 -12514.294} C_VEL
LIN {X 0,Y 376.028,Z 589.932,A -85,B 0,C 180,E1 -12515.9,E2 -12515.9} C_VEL
LIN {X 0,Y 376.677,Z 583.561,A -85,B 0,C 180,E1 -12517.505,E2 -12517.505} C_VEL
LIN {X 0,Y 377.473,Z 574.74,A -85,B 0,C 180,E1 -12519.323,E2 -12519.323} C_VEL
LIN {X 0,Y 378.312,Z 568.009,A -85,B 0,C 180,E1 -12520.484,E2 -12520.484} C_VEL
LIN {X 0,Y 378.11,Z 564.008,A -85,B 0,C 180,E1 -12521.144,E2 -12521.144} C_VEL
LIN {X 0,Y 376.105,Z 557.339,A -85,B 0,C 180,E1 -12522.22,E2 -12522.22} C_VEL
LIN {X 0,Y 374.16,Z 550.219,A -85,B 0,C 180,E1 -12523.23,E2 -12523.23} C_VEL
LIN {X 0,Y 374.035,Z 545.516,A -85,B 0,C 180,E1 -12523.775,E2 -12523.775} C_VEL
LIN {X 0,Y 375.154,Z 533.717,A -85,B 0,C 180,E1 -12524.927,E2 -12524.927} C_VEL
LIN {X 0,Y 376.209,Z 521.896,A -85,B 0,C 180,E1 -12525.855,E2 -12525.855} C_VEL
LIN {X 0,Y 377.186,Z 508.981,A -85,B 0,C 180,E1 -12526.647,E2 -12526.647} C_VEL
LIN {X 0,Y 377.926,Z 495.116,A -85,B 0,C 180,E1 -12527.275,E2 -12527.275} C_VEL
LIN {X 0,Y 378.407,Z 482.137,A -85,B 0,C 180,E1 -12527.671,E2 -12527.671} C_VEL
LIN {X 0,Y 380.401,Z 377.449,A -85,B 0,C 180,E1 -12529.661,E2 -12529.661} C_VEL
LIN {X 0,Y 377.818,Z 365.373,A -85,B 0,C 180,E1 -12530.072,E2 -12530.072} C_VEL
LIN {X 0,Y 371.029,Z 347.819,A -85,B 0,C 180,E1 -12530.918,E2 -12530.918} C_VEL
LIN {X 0,Y 368.947,Z 338.155,A -85,B 0,C 180,E1 -12533.468,E2 -12533.468} C_VEL
LIN {X 0,Y 368.882,Z 338.165,A -85,B 0,C 180,E1 -12536.432,E2 -12536.432} C_VEL
LIN {X 0,Y 368.894,Z 338.155,A -85,B 0,C 180,E1 -12539.692,E2 -12539.692} C_VEL
LIN {X 0,Y 368.897,Z 338.158,A -85,B 0,C 180,E1 -12543.538,E2 -12543.538} C_VEL
LIN {X 0,Y 368.897,Z 338.158,A -85,B 0,C 180,E1 -12546.854,E2 -12546.854} C_VEL
LIN {X 0,Y 368.886,Z 338.16,A -85,B 0,C 180,E1 -12550.374,E2 -12550.374} C_VEL
LIN {X 0,Y 368.881,Z 338.159,A -85,B 0,C 180,E1 -12553.615,E2 -12553.615} C_VEL
LIN {X 0,Y 368.886,Z 338.163,A -85,B 0,C 180,E1 -12556.695,E2 -12556.695} C_VEL
LIN {X 0,Y 368.887,Z 338.156,A -85,B 0,C 180,E1 -12559.648,E2 -12559.648} C_VEL
LIN {X 0,Y 368.9,Z 338.154,A -85,B 0,C 180,E1 -12563.145,E2 -12563.145} C_VEL
LIN {X 0,Y 368.898,Z 338.154,A -85,B 0,C 180,E1 -12566.462,E2 -12566.462} C_VEL
LIN {X 0,Y 368.898,Z 338.157,A -85,B 0,C 180,E1 -12569.043,E2 -12569.043} C_VEL
LIN {X 0,Y 368.909,Z 338.151,A -85,B 0,C 180,E1 -12571.558,E2 -12571.558} C_VEL
LIN {X 0,Y 368.889,Z 338.157,A -85,B 0,C 180,E1 -12575.219,E2 -12575.219} C_VEL
LIN {X 0,Y 368.922,Z 338.148,A -85,B 0,C 180,E1 -12577.604,E2 -12577.604} C_VEL
LIN {X 0,Y 368.918,Z 338.143,A -85,B 0,C 180,E1 -12581.103,E2 -12581.103} C_VEL
LIN {X 0,Y 368.943,Z 338.153,A -85,B 0,C 180,E1 -12584.532,E2 -12584.532} C_VEL
LIN {X 0,Y 369.061,Z 338.126,A -85,B 0,C 180,E1 -12586.79,E2 -12586.79} C_VEL
LIN {X 0,Y 369.066,Z 338.115,A -85,B 0,C 180,E1 -12590.131,E2 -12590.131} C_VEL
LIN {X 0,Y 369.163,Z 338.123,A -85,B 0,C 180,E1 -12593.441,E2 -12593.441} C_VEL
LIN {X 0,Y 369.312,Z 338.105,A -85,B 0,C 180,E1 -12597.818,E2 -12597.818} C_VEL
LIN {X 0,Y 369.238,Z 338.107,A -85,B 0,C 180,E1 -12601.09,E2 -12601.09} C_VEL
LIN {X 0,Y 369.305,Z 338.107,A -85,B 0,C 180,E1 -12602.181,E2 -12602.181} C_VEL
LIN {X 0,Y 369.164,Z 338.123,A -85,B 0,C 180,E1 -12606.559,E2 -12606.559} C_VEL
LIN {X 0,Y 369.066,Z 338.135,A -85,B 0,C 180,E1 -12609.868,E2 -12609.868} C_VEL
LIN {X 0,Y 369.04,Z 338.14,A -85,B 0,C 180,E1 -12613.772,E2 -12613.772} C_VEL
LIN {X 0,Y 369.004,Z 338.144,A -85,B 0,C 180,E1 -12617.768,E2 -12617.768} C_VEL
LIN {X 0,Y 368.93,Z 338.153,A -85,B 0,C 180,E1 -12621.219,E2 -12621.219} C_VEL
LIN {X 0,Y 368.944,Z 338.15,A -85,B 0,C 180,E1 -12624.776,E2 -12624.776} C_VEL
LIN {X 0,Y 368.961,Z 338.148,A -85,B 0,C 180,E1 -12628.437,E2 -12628.437} C_VEL
LIN {X 0,Y 368.9,Z 338.156,A -85,B 0,C 180,E1 -12632.238,E2 -12632.238} C_VEL
LIN {X 0,Y 368.931,Z 338.155,A -85,B 0,C 180,E1 -12635.001,E2 -12635.001} C_VEL
LIN {X 0,Y 368.912,Z 338.154,A -85,B 0,C 180,E1 -12638.64,E2 -12638.64} C_VEL
LIN {X 0,Y 368.883,Z 338.162,A -85,B 0,C 180,E1 -12642.009,E2 -12642.009} C_VEL
LIN {X 0,Y 368.881,Z 338.163,A -85,B 0,C 180,E1 -12645.176,E2 -12645.176} C_VEL
LIN {X 0,Y 368.883,Z 338.16,A -85,B 0,C 180,E1 -12648.177,E2 -12648.177} C_VEL
LIN {X 0,Y 368.911,Z 338.161,A -85,B 0,C 180,E1 -12651.359,E2 -12651.359} C_VEL
LIN {X 0,Y 368.938,Z 338.159,A -85,B 0,C 180,E1 -12655.146,E2 -12655.146} C_VEL
LIN {X 0,Y 368.938,Z 338.246,A -85,B 0,C 180,E1 -12657.873,E2 -12657.873} C_VEL
LIN {X 0,Y 372.217,Z 352.335,A -85,B 0,C 180,E1 -12661.218,E2 -12661.218} C_VEL
LIN {X 0,Y 373.933,Z 361.011,A -85,B 0,C 180,E1 -12663.187,E2 -12663.187} C_VEL
LIN {X 0,Y 373.73,Z 366.125,A -85,B 0,C 180,E1 -12664.252,E2 -12664.252} C_VEL
LIN {X 0,Y 373.727,Z 366.851,A -85,B 0,C 180,E1 -12664.327,E2 -12664.327} C_VEL
LIN {X 0,Y 379.902,Z 402.171,A -85,B 0,C 180,E1 -12665.443,E2 -12665.443} C_VEL
LIN {X 0,Y 378.759,Z 474.499,A -85,B 0,C 180,E1 -12666.82,E2 -12666.82} C_VEL
LIN {X 0,Y 378.082,Z 504.937,A -85,B 0,C 180,E1 -12667.42,E2 -12667.42} C_VEL
LIN {X 0,Y 377.331,Z 519.49,A -85,B 0,C 180,E1 -12667.914,E2 -12667.914} C_VEL
LIN {X 0,Y 376.303,Z 534.009,A -85,B 0,C 180,E1 -12668.642,E2 -12668.642} C_VEL
LIN {X 0,Y 375.256,Z 546.208,A -85,B 0,C 180,E1 -12669.46,E2 -12669.46} C_VEL
LIN {X 0,Y 374.098,Z 558.684,A -85,B 0,C 180,E1 -12670.521,E2 -12670.521} C_VEL
LIN {X 0,Y 372.783,Z 570.248,A -85,B 0,C 180,E1 -12671.734,E2 -12671.734} C_VEL
LIN {X 0,Y 371.644,Z 579.873,A -85,B 0,C 180,E1 -12672.955,E2 -12672.955} C_VEL
LIN {X 0,Y 370.392,Z 590.573,A -85,B 0,C 180,E1 -12674.595,E2 -12674.595} C_VEL
LIN {X 0,Y 369.522,Z 599.904,A -85,B 0,C 180,E1 -12676.348,E2 -12676.348} C_VEL
LIN {X 0,Y 368.658,Z 607.869,A -85,B 0,C 180,E1 -12678.174,E2 -12678.174} C_VEL
LIN {X 0,Y 368.032,Z 614.667,A -85,B 0,C 180,E1 -12680.104,E2 -12680.104} C_VEL
LIN {X 0,Y 367.653,Z 620.693,A -85,B 0,C 180,E1 -12682.31,E2 -12682.31} C_VEL
LIN {X 0,Y 367.464,Z 625.109,A -85,B 0,C 180,E1 -12684.513,E2 -12684.513} C_VEL
LIN {X 0,Y 367.375,Z 628.061,A -85,B 0,C 180,E1 -12686.71,E2 -12686.71} C_VEL
LIN {X 0,Y 367.417,Z 629.636,A -85,B 0,C 180,E1 -12688.904,E2 -12688.904} C_VEL
LIN {X 0,Y 367.415,Z 629.865,A -85,B 0,C 180,E1 -12691.096,E2 -12691.096} C_VEL
LIN {X 0,Y 367.371,Z 628.762,A -85,B 0,C 180,E1 -12693.29,E2 -12693.29} C_VEL
LIN {X 0,Y 367.448,Z 626.312,A -85,B 0,C 180,E1 -12695.488,E2 -12695.488} C_VEL
LIN {X 0,Y 367.673,Z 622.455,A -85,B 0,C 180,E1 -12697.69,E2 -12697.69} C_VEL
LIN {X 0,Y 368.111,Z 617.038,A -85,B 0,C 180,E1 -12699.894,E2 -12699.894} C_VEL
LIN {X 0,Y 368.663,Z 611.882,A -85,B 0,C 180,E1 -12701.547,E2 -12701.547} C_VEL
LIN {X 0,Y 369.59,Z 604.527,A -85,B 0,C 180,E1 -12703.466,E2 -12703.466} C_VEL
LIN {X 0,Y 370.549,Z 596.798,A -85,B 0,C 180,E1 -12705.117,E2 -12705.117} C_VEL
LIN {X 0,Y 371.839,Z 587.563,A -85,B 0,C 180,E1 -12706.752,E2 -12706.752} C_VEL
LIN {X 0,Y 373.308,Z 577.377,A -85,B 0,C 180,E1 -12708.24,E2 -12708.24} C_VEL
LIN {X 0,Y 374.859,Z 566.186,A -85,B 0,C 180,E1 -12709.58,E2 -12709.58} C_VEL
LIN {X 0,Y 376.353,Z 553.838,A -85,B 0,C 180,E1 -12710.782,E2 -12710.782} C_VEL
LIN {X 0,Y 377.595,Z 541.956,A -85,B 0,C 180,E1 -12711.712,E2 -12711.712} C_VEL
LIN {X 0,Y 378.767,Z 529.027,A -85,B 0,C 180,E1 -12712.501,E2 -12712.501} C_VEL
LIN {X 0,Y 379.861,Z 515.147,A -85,B 0,C 180,E1 -12713.115,E2 -12713.115} C_VEL
LIN {X 0,Y 380.583,Z 500.741,A -85,B 0,C 180,E1 -12713.537,E2 -12713.537} C_VEL
LIN {X 0,Y 382.645,Z 404.036,A -85,B 0,C 180,E1 -12715.386,E2 -12715.386} C_VEL
LIN {X 0,Y 379.209,Z 385.166,A -85,B 0,C 180,E1 -12716.047,E2 -12716.047} C_VEL
LIN {X 0,Y 375.161,Z 366.165,A -85,B 0,C 180,E1 -12716.793,E2 -12716.793} C_VEL
LIN {X 0,Y 374.145,Z 359.606,A -85,B 0,C 180,E1 -12718.313,E2 -12718.313} C_VEL
LIN {X 0,Y 371.076,Z 346.518,A -85,B 0,C 180,E1 -12721.54,E2 -12721.54} C_VEL
LIN {X 0,Y 368.931,Z 338.153,A -85,B 0,C 180,E1 -12723.74,E2 -12723.74} C_VEL
LIN {X 0,Y 368.904,Z 338.157,A -85,B 0,C 180,E1 -12727.563,E2 -12727.563} C_VEL
LIN {X 0,Y 368.912,Z 338.159,A -85,B 0,C 180,E1 -12730.37,E2 -12730.37} C_VEL
LIN {X 0,Y 368.883,Z 338.156,A -85,B 0,C 180,E1 -12733.616,E2 -12733.616} C_VEL
LIN {X 0,Y 368.887,Z 338.161,A -85,B 0,C 180,E1 -12736.696,E2 -12736.696} C_VEL
LIN {X 0,Y 368.914,Z 338.155,A -85,B 0,C 180,E1 -12739.643,E2 -12739.643} C_VEL
LIN {X 0,Y 368.903,Z 338.153,A -85,B 0,C 180,E1 -12743.145,E2 -12743.145} C_VEL
LIN {X 0,Y 368.899,Z 338.155,A -85,B 0,C 180,E1 -12746.462,E2 -12746.462} C_VEL
LIN {X 0,Y 368.931,Z 338.152,A -85,B 0,C 180,E1 -12749.047,E2 -12749.047} C_VEL
LIN {X 0,Y 368.88,Z 338.157,A -85,B 0,C 180,E1 -12752.79,E2 -12752.79} C_VEL
LIN {X 0,Y 368.931,Z 338.157,A -85,B 0,C 180,E1 -12756.119,E2 -12756.119} C_VEL
LIN {X 0,Y 368.94,Z 338.154,A -85,B 0,C 180,E1 -12759.947,E2 -12759.947} C_VEL
LIN {X 0,Y 368.979,Z 338.143,A -85,B 0,C 180,E1 -12763.399,E2 -12763.399} C_VEL
LIN {X 0,Y 369.061,Z 338.128,A -85,B 0,C 180,E1 -12766.791,E2 -12766.791} C_VEL
LIN {X 0,Y 369.066,Z 338.136,A -85,B 0,C 180,E1 -12770.132,E2 -12770.132} C_VEL
LIN {X 0,Y 369.164,Z 338.122,A -85,B 0,C 180,E1 -12773.441,E2 -12773.441} C_VEL
LIN {X 0,Y 369.306,Z 338.102,A -85,B 0,C 180,E1 -12777.819,E2 -12777.819} C_VEL
LIN {X 0,Y 369.207,Z 338.114,A -85,B 0,C 180,E1 -12781.091,E2 -12781.091} C_VEL
LIN {X 0,Y 369.312,Z 338.1,A -85,B 0,C 180,E1 -12782.182,E2 -12782.182} C_VEL
LIN {X 0,Y 369.162,Z 338.114,A -85,B 0,C 180,E1 -12786.559,E2 -12786.559} C_VEL
LIN {X 0,Y 369.066,Z 338.137,A -85,B 0,C 180,E1 -12789.869,E2 -12789.869} C_VEL
LIN {X 0,Y 369.041,Z 338.143,A -85,B 0,C 180,E1 -12793.773,E2 -12793.773} C_VEL
LIN {X 0,Y 368.957,Z 338.15,A -85,B 0,C 180,E1 -12797.745,E2 -12797.745} C_VEL
LIN {X 0,Y 368.912,Z 338.149,A -85,B 0,C 180,E1 -12801.221,E2 -12801.221} C_VEL
LIN {X 0,Y 368.911,Z 338.153,A -85,B 0,C 180,E1 -12803.874,E2 -12803.874} C_VEL
LIN {X 0,Y 368.86,Z 338.164,A -85,B 0,C 180,E1 -12807.212,E2 -12807.212} C_VEL
LIN {X 0,Y 368.895,Z 338.135,A -85,B 0,C 180,E1 -12809.693,E2 -12809.693} C_VEL
LIN {X 0,Y 368.898,Z 338.161,A -85,B 0,C 180,E1 -12813.538,E2 -12813.538} C_VEL
LIN {X 0,Y 368.898,Z 338.139,A -85,B 0,C 180,E1 -12816.854,E2 -12816.854} C_VEL
LIN {X 0,Y 368.886,Z 338.155,A -85,B 0,C 180,E1 -12820.374,E2 -12820.374} C_VEL
LIN {X 0,Y 368.882,Z 338.164,A -85,B 0,C 180,E1 -12823.615,E2 -12823.615} C_VEL
LIN {X 0,Y 368.886,Z 338.156,A -85,B 0,C 180,E1 -12826.695,E2 -12826.695} C_VEL
LIN {X 0,Y 368.887,Z 338.156,A -85,B 0,C 180,E1 -12829.648,E2 -12829.648} C_VEL
LIN {X 0,Y 368.897,Z 338.161,A -85,B 0,C 180,E1 -12833.146,E2 -12833.146} C_VEL
LIN {X 0,Y 368.933,Z 338.184,A -85,B 0,C 180,E1 -12835.146,E2 -12835.146} C_VEL
LIN {X 0,Y 371.285,Z 348.205,A -85,B 0,C 180,E1 -12837.946,E2 -12837.946} C_VEL
LIN {X 0,Y 380.951,Z 370.137,A -85,B 0,C 180,E1 -12839.216,E2 -12839.216} C_VEL
LIN {X 0,Y 382.285,Z 374.653,A -85,B 0,C 180,E1 -12839.416,E2 -12839.416} C_VEL
LIN {X 0,Y 383.161,Z 379.29,A -85,B 0,C 180,E1 -12839.581,E2 -12839.581} C_VEL
LIN {X 0,Y 380.896,Z 484.083,A -85,B 0,C 180,E1 -12841.595,E2 -12841.595} C_VEL
LIN {X 0,Y 380.195,Z 498.306,A -85,B 0,C 180,E1 -12842.064,E2 -12842.064} C_VEL
LIN {X 0,Y 379.181,Z 511.722,A -85,B 0,C 180,E1 -12842.709,E2 -12842.709} C_VEL
LIN {X 0,Y 378.111,Z 524.086,A -85,B 0,C 180,E1 -12843.507,E2 -12843.507} C_VEL
LIN {X 0,Y 376.697,Z 537.177,A -85,B 0,C 180,E1 -12844.589,E2 -12844.589} C_VEL
LIN {X 0,Y 375.168,Z 549.002,A -85,B 0,C 180,E1 -12845.809,E2 -12845.809} C_VEL
LIN {X 0,Y 373.806,Z 560.219,A -85,B 0,C 180,E1 -12847.246,E2 -12847.246} C_VEL
LIN {X 0,Y 372.453,Z 569.635,A -85,B 0,C 180,E1 -12848.701,E2 -12848.701} C_VEL
LIN {X 0,Y 371.133,Z 578.534,A -85,B 0,C 180,E1 -12850.359,E2 -12850.359} C_VEL
LIN {X 0,Y 369.971,Z 587.034,A -85,B 0,C 180,E1 -12852.306,E2 -12852.306} C_VEL
LIN {X 0,Y 369.105,Z 592.942,A -85,B 0,C 180,E1 -12853.973,E2 -12853.973} C_VEL
LIN {X 0,Y 368.366,Z 599.227,A -85,B 0,C 180,E1 -12856.203,E2 -12856.203} C_VEL
LIN {X 0,Y 367.898,Z 602.804,A -85,B 0,C 180,E1 -12857.87,E2 -12857.87} C_VEL
LIN {X 0,Y 367.533,Z 606.288,A -85,B 0,C 180,E1 -12860.09,E2 -12860.09} C_VEL
LIN {X 0,Y 367.417,Z 608.366,A -85,B 0,C 180,E1 -12862.305,E2 -12862.305} C_VEL
LIN {X 0,Y 367.427,Z 609.103,A -85,B 0,C 180,E1 -12864.512,E2 -12864.512} C_VEL
LIN {X 0,Y 367.389,Z 608.524,A -85,B 0,C 180,E1 -12866.71,E2 -12866.71} C_VEL
LIN {X 0,Y 367.495,Z 606.615,A -85,B 0,C 180,E1 -12868.904,E2 -12868.904} C_VEL
LIN {X 0,Y 367.645,Z 603.33,A -85,B 0,C 180,E1 -12871.095,E2 -12871.095} C_VEL
LIN {X 0,Y 368.062,Z 598.577,A -85,B 0,C 180,E1 -12873.284,E2 -12873.284} C_VEL
LIN {X 0,Y 368.75,Z 592.209,A -85,B 0,C 180,E1 -12875.468,E2 -12875.468} C_VEL
LIN {X 0,Y 369.406,Z 586.235,A -85,B 0,C 180,E1 -12877.104,E2 -12877.104} C_VEL
LIN {X 0,Y 370.323,Z 577.677,A -85,B 0,C 180,E1 -12879.019,E2 -12879.019} C_VEL
LIN {X 0,Y 370.873,Z 572.036,A -85,B 0,C 180,E1 -12880.095,E2 -12880.095} C_VEL
LIN {X 0,Y 372.252,Z 561.954,A -85,B 0,C 180,E1 -12881.71,E2 -12881.71} C_VEL
LIN {X 0,Y 373.456,Z 550.689,A -85,B 0,C 180,E1 -12883.19,E2 -12883.19} C_VEL
LIN {X 0,Y 374.035,Z 545.516,A -85,B 0,C 180,E1 -12883.775,E2 -12883.775} C_VEL
LIN {X 0,Y 373.904,Z 540.773,A -85,B 0,C 180,E1 -12884.301,E2 -12884.301} C_VEL
LIN {X 0,Y 371.916,Z 532.898,A -85,B 0,C 180,E1 -12885.172,E2 -12885.172} C_VEL
LIN {X 0,Y 369.915,Z 524.734,A -85,B 0,C 180,E1 -12885.984,E2 -12885.984} C_VEL
LIN {X 0,Y 369.72,Z 519.402,A -85,B 0,C 180,E1 -12886.397,E2 -12886.397} C_VEL
LIN {X 0,Y 370.677,Z 506.438,A -85,B 0,C 180,E1 -12887.161,E2 -12887.161} C_VEL
LIN {X 0,Y 371.425,Z 492.354,A -85,B 0,C 180,E1 -12887.765,E2 -12887.765} C_VEL
LIN {X 0,Y 371.907,Z 477.402,A -85,B 0,C 180,E1 -12888.168,E2 -12888.168} C_VEL
LIN {X 0,Y 373.794,Z 377.814,A -85,B 0,C 180,E1 -12890.083,E2 -12890.083} C_VEL
LIN {X 0,Y 371.357,Z 367.209,A -85,B 0,C 180,E1 -12890.464,E2 -12890.464} C_VEL
LIN {X 0,Y 363.884,Z 348.095,A -85,B 0,C 180,E1 -12891.401,E2 -12891.401} C_VEL
LIN {X 0,Y 361.891,Z 339.034,A -85,B 0,C 180,E1 -12893.87,E2 -12893.87} C_VEL
LIN {X 0,Y 361.837,Z 339.04,A -85,B 0,C 180,E1 -12897.785,E2 -12897.785} C_VEL
LIN {X 0,Y 361.829,Z 339.041,A -85,B 0,C 180,E1 -12901.28,E2 -12901.28} C_VEL
LIN {X 0,Y 361.853,Z 339.037,A -85,B 0,C 180,E1 -12904.281,E2 -12904.281} C_VEL
LIN {X 0,Y 361.859,Z 339.036,A -85,B 0,C 180,E1 -12907.221,E2 -12907.221} C_VEL
LIN {X 0,Y 361.813,Z 339.043,A -85,B 0,C 180,E1 -12910.75,E2 -12910.75} C_VEL
LIN {X 0,Y 361.814,Z 339.041,A -85,B 0,C 180,E1 -12914.369,E2 -12914.369} C_VEL
LIN {X 0,Y 361.825,Z 339.036,A -85,B 0,C 180,E1 -12917.57,E2 -12917.57} C_VEL
LIN {X 0,Y 361.843,Z 339.034,A -85,B 0,C 180,E1 -12921.572,E2 -12921.572} C_VEL
LIN {X 0,Y 361.876,Z 339.036,A -85,B 0,C 180,E1 -12924.655,E2 -12924.655} C_VEL
LIN {X 0,Y 361.84,Z 339.033,A -85,B 0,C 180,E1 -12928.37,E2 -12928.37} C_VEL
LIN {X 0,Y 361.851,Z 339.032,A -85,B 0,C 180,E1 -12930.95,E2 -12930.95} C_VEL
LIN {X 0,Y 361.863,Z 339.036,A -85,B 0,C 180,E1 -12934.705,E2 -12934.705} C_VEL
LIN {X 0,Y 361.863,Z 339.018,A -85,B 0,C 180,E1 -12938.345,E2 -12938.345} C_VEL
LIN {X 0,Y 361.907,Z 339.02,A -85,B 0,C 180,E1 -12942.092,E2 -12942.092} C_VEL
LIN {X 0,Y 361.983,Z 339.015,A -85,B 0,C 180,E1 -12946.113,E2 -12946.113} C_VEL
LIN {X 0,Y 362.003,Z 338.992,A -85,B 0,C 180,E1 -12949.937,E2 -12949.937} C_VEL
LIN {X 0,Y 362.126,Z 338.999,A -85,B 0,C 180,E1 -12953.313,E2 -12953.313} C_VEL
LIN {X 0,Y 362.274,Z 338.981,A -85,B 0,C 180,E1 -12957.776,E2 -12957.776} C_VEL
LIN {X 0,Y 362.207,Z 338.983,A -85,B 0,C 180,E1 -12961.111,E2 -12961.111} C_VEL
LIN {X 0,Y 362.268,Z 338.984,A -85,B 0,C 180,E1 -12962.223,E2 -12962.223} C_VEL
LIN {X 0,Y 362.127,Z 338.999,A -85,B 0,C 180,E1 -12966.687,E2 -12966.687} C_VEL
LIN {X 0,Y 362.003,Z 339.014,A -85,B 0,C 180,E1 -12970.063,E2 -12970.063} C_VEL
LIN {X 0,Y 362.001,Z 339.015,A -85,B 0,C 180,E1 -12973.899,E2 -12973.899} C_VEL
LIN {X 0,Y 361.97,Z 339.019,A -85,B 0,C 180,E1 -12977.938,E2 -12977.938} C_VEL
LIN {X 0,Y 361.893,Z 339.03,A -85,B 0,C 180,E1 -12981.653,E2 -12981.653} C_VEL
LIN {X 0,Y 361.907,Z 339.029,A -85,B 0,C 180,E1 -12985.291,E2 -12985.291} C_VEL
LIN {X 0,Y 361.876,Z 339.031,A -85,B 0,C 180,E1 -12989.079,E2 -12989.079} C_VEL
LIN {X 0,Y 361.85,Z 339.034,A -85,B 0,C 180,E1 -12992.944,E2 -12992.944} C_VEL
LIN {X 0,Y 361.87,Z 339.035,A -85,B 0,C 180,E1 -12995.636,E2 -12995.636} C_VEL
LIN {X 0,Y 361.872,Z 339.032,A -85,B 0,C 180,E1 -12999.027,E2 -12999.027} C_VEL
LIN {X 0,Y 361.837,Z 339.039,A -85,B 0,C 180,E1 -13002.828,E2 -13002.828} C_VEL
LIN {X 0,Y 361.819,Z 339.041,A -85,B 0,C 180,E1 -13005.946,E2 -13005.946} C_VEL
LIN {X 0,Y 361.837,Z 339.041,A -85,B 0,C 180,E1 -13009.244,E2 -13009.244} C_VEL
LIN {X 0,Y 361.866,Z 339.039,A -85,B 0,C 180,E1 -13012.777,E2 -13012.777} C_VEL
LIN {X 0,Y 361.856,Z 339.041,A -85,B 0,C 180,E1 -13015.72,E2 -13015.72} C_VEL
LIN {X 0,Y 361.892,Z 339.142,A -85,B 0,C 180,E1 -13017.473,E2 -13017.473} C_VEL
LIN {X 0,Y 364.931,Z 352.228,A -85,B 0,C 180,E1 -13020.661,E2 -13020.661} C_VEL
LIN {X 0,Y 367.126,Z 363.454,A -85,B 0,C 180,E1 -13023.265,E2 -13023.265} C_VEL
LIN {X 0,Y 366.976,Z 366.211,A -85,B 0,C 180,E1 -13023.847,E2 -13023.847} C_VEL
LIN {X 0,Y 373.333,Z 403.128,A -85,B 0,C 180,E1 -13025.045,E2 -13025.045} C_VEL
LIN {X 0,Y 371.921,Z 486.517,A -85,B 0,C 180,E1 -13026.657,E2 -13026.657} C_VEL
LIN {X 0,Y 371.335,Z 506.961,A -85,B 0,C 180,E1 -13027.097,E2 -13027.097} C_VEL
LIN {X 0,Y 370.543,Z 521.547,A -85,B 0,C 180,E1 -13027.634,E2 -13027.634} C_VEL
LIN {X 0,Y 369.474,Z 535.48,A -85,B 0,C 180,E1 -13028.374,E2 -13028.374} C_VEL
LIN {X 0,Y 368.351,Z 548.485,A -85,B 0,C 180,E1 -13029.299,E2 -13029.299} C_VEL
LIN {X 0,Y 367.052,Z 560.953,A -85,B 0,C 180,E1 -13030.423,E2 -13030.423} C_VEL
LIN {X 0,Y 365.583,Z 573.16,A -85,B 0,C 180,E1 -13031.797,E2 -13031.797} C_VEL
LIN {X 0,Y 364.365,Z 583.255,A -85,B 0,C 180,E1 -13033.182,E2 -13033.182} C_VEL
LIN {X 0,Y 363.095,Z 593.295,A -85,B 0,C 180,E1 -13034.853,E2 -13034.853} C_VEL
LIN {X 0,Y 362.335,Z 601.638,A -85,B 0,C 180,E1 -13036.541,E2 -13036.541} C_VEL
LIN {X 0,Y 361.433,Z 609.6,A -85,B 0,C 180,E1 -13038.503,E2 -13038.503} C_VEL
LIN {X 0,Y 360.851,Z 616,A -85,B 0,C 180,E1 -13040.471,E2 -13040.471} C_VEL
LIN {X 0,Y 360.524,Z 621.665,A -85,B 0,C 180,E1 -13042.72,E2 -13042.72} C_VEL
LIN {X 0,Y 360.381,Z 624.85,A -85,B 0,C 180,E1 -13044.404,E2 -13044.404} C_VEL
LIN {X 0,Y 360.295,Z 627.824,A -85,B 0,C 180,E1 -13046.645,E2 -13046.645} C_VEL
LIN {X 0,Y 360.318,Z 629.419,A -85,B 0,C 180,E1 -13048.882,E2 -13048.882} C_VEL
LIN {X 0,Y 360.358,Z 629.712,A -85,B 0,C 180,E1 -13050,E2 -13050} C_VEL
LIN {X 0,Y 360.26,Z 629.293,A -85,B 0,C 180,E1 -13052.236,E2 -13052.236} C_VEL
LIN {X 0,Y 360.332,Z 627.542,A -85,B 0,C 180,E1 -13054.475,E2 -13054.475} C_VEL
LIN {X 0,Y 360.492,Z 624.421,A -85,B 0,C 180,E1 -13056.718,E2 -13056.718} C_VEL
LIN {X 0,Y 360.802,Z 619.838,A -85,B 0,C 180,E1 -13058.965,E2 -13058.965} C_VEL
LIN {X 0,Y 361.226,Z 615.318,A -85,B 0,C 180,E1 -13060.651,E2 -13060.651} C_VEL
LIN {X 0,Y 362.124,Z 608.826,A -85,B 0,C 180,E1 -13062.612,E2 -13062.612} C_VEL
LIN {X 0,Y 363.048,Z 600.783,A -85,B 0,C 180,E1 -13064.576,E2 -13064.576} C_VEL
LIN {X 0,Y 364.293,Z 592.383,A -85,B 0,C 180,E1 -13066.245,E2 -13066.245} C_VEL
LIN {X 0,Y 365.803,Z 582.287,A -85,B 0,C 180,E1 -13067.903,E2 -13067.903} C_VEL
LIN {X 0,Y 367.536,Z 571.005,A -85,B 0,C 180,E1 -13069.405,E2 -13069.405} C_VEL
LIN {X 0,Y 369.043,Z 559.812,A -85,B 0,C 180,E1 -13070.629,E2 -13070.629} C_VEL
LIN {X 0,Y 370.407,Z 548.087,A -85,B 0,C 180,E1 -13071.676,E2 -13071.676} C_VEL
LIN {X 0,Y 371.731,Z 535.216,A -85,B 0,C 180,E1 -13072.584,E2 -13072.584} C_VEL
LIN {X 0,Y 372.91,Z 522.178,A -85,B 0,C 180,E1 -13073.278,E2 -13073.278} C_VEL
LIN {X 0,Y 373.84,Z 508.193,A -85,B 0,C 180,E1 -13073.804,E2 -13073.804} C_VEL
LIN {X 0,Y 374.419,Z 490.643,A -85,B 0,C 180,E1 -13074.206,E2 -13074.206} C_VEL
LIN {X 0,Y 376.27,Z 404.249,A -85,B 0,C 180,E1 -13075.879,E2 -13075.879} C_VEL
LIN {X 0,Y 371.254,Z 378.17,A -85,B 0,C 180,E1 -13076.846,E2 -13076.846} C_VEL
LIN {X 0,Y 368.794,Z 367.839,A -85,B 0,C 180,E1 -13077.28,E2 -13077.28} C_VEL
LIN {X 0,Y 368.189,Z 365.885,A -85,B 0,C 180,E1 -13077.403,E2 -13077.403} C_VEL
LIN {X 0,Y 365.801,Z 354.609,A -85,B 0,C 180,E1 -13080.167,E2 -13080.167} C_VEL
LIN {X 0,Y 362.84,Z 342.72,A -85,B 0,C 180,E1 -13083.255,E2 -13083.255} C_VEL
LIN {X 0,Y 361.873,Z 339.035,A -85,B 0,C 180,E1 -13084.279,E2 -13084.279} C_VEL
LIN {X 0,Y 361.864,Z 339.036,A -85,B 0,C 180,E1 -13087.223,E2 -13087.223} C_VEL
LIN {X 0,Y 361.837,Z 339.039,A -85,B 0,C 180,E1 -13090.756,E2 -13090.756} C_VEL
LIN {X 0,Y 361.819,Z 339.041,A -85,B 0,C 180,E1 -13094.369,E2 -13094.369} C_VEL
LIN {X 0,Y 361.838,Z 339.035,A -85,B 0,C 180,E1 -13097.568,E2 -13097.568} C_VEL
LIN {X 0,Y 361.872,Z 339.03,A -85,B 0,C 180,E1 -13100.974,E2 -13100.974} C_VEL
LIN {X 0,Y 361.876,Z 339.034,A -85,B 0,C 180,E1 -13104.656,E2 -13104.656} C_VEL
LIN {X 0,Y 361.84,Z 339.04,A -85,B 0,C 180,E1 -13108.371,E2 -13108.371} C_VEL
LIN {X 0,Y 361.867,Z 339.032,A -85,B 0,C 180,E1 -13110.953,E2 -13110.953} C_VEL
LIN {X 0,Y 361.896,Z 339.03,A -85,B 0,C 180,E1 -13114.708,E2 -13114.708} C_VEL
LIN {X 0,Y 361.863,Z 339.03,A -85,B 0,C 180,E1 -13118.346,E2 -13118.346} C_VEL
LIN {X 0,Y 361.97,Z 339.015,A -85,B 0,C 180,E1 -13122.062,E2 -13122.062} C_VEL
LIN {X 0,Y 362.001,Z 339.011,A -85,B 0,C 180,E1 -13126.101,E2 -13126.101} C_VEL
LIN {X 0,Y 362.031,Z 339.014,A -85,B 0,C 180,E1 -13129.938,E2 -13129.938} C_VEL
LIN {X 0,Y 362.127,Z 338.998,A -85,B 0,C 180,E1 -13133.313,E2 -13133.313} C_VEL
LIN {X 0,Y 362.269,Z 338.978,A -85,B 0,C 180,E1 -13137.777,E2 -13137.777} C_VEL
LIN {X 0,Y 362.178,Z 338.989,A -85,B 0,C 180,E1 -13141.112,E2 -13141.112} C_VEL
LIN {X 0,Y 362.275,Z 338.976,A -85,B 0,C 180,E1 -13142.224,E2 -13142.224} C_VEL
LIN {X 0,Y 362.125,Z 338.99,A -85,B 0,C 180,E1 -13146.687,E2 -13146.687} C_VEL
LIN {X 0,Y 362.003,Z 339.015,A -85,B 0,C 180,E1 -13150.063,E2 -13150.063} C_VEL
LIN {X 0,Y 361.983,Z 339.022,A -85,B 0,C 180,E1 -13153.887,E2 -13153.887} C_VEL
LIN {X 0,Y 361.887,Z 339.032,A -85,B 0,C 180,E1 -13158.103,E2 -13158.103} C_VEL
LIN {X 0,Y 361.856,Z 339.032,A -85,B 0,C 180,E1 -13161.656,E2 -13161.656} C_VEL
LIN {X 0,Y 361.863,Z 339.029,A -85,B 0,C 180,E1 -13165.295,E2 -13165.295} C_VEL
